(* POU Device/Valve/fbWaterSupplyValve, ST *)
FUNCTION_BLOCK fbWaterSupplyValve
VAR_INPUT
	xManualMode:			BOOL;
	wOffDelay:				WORD:=3;
	xStopSupplying:		BOOL;
	rWaterLevel:			REAL;
	rWaterLevelNotOK:	REAL;
	xUpperLevel:			BOOL;
	xOnAutoWorking:		BOOL;
	xSensor:				BOOL;
END_VAR
VAR_IN_OUT

	xOnManual:			BOOL;

END_VAR
VAR_OUTPUT
	xDO_On:				BOOL;
	xState:					BOOL;
END_VAR
VAR
	tfOffDelay:				TOF;
	xDO_OnOld:			BOOL;
	tnDelayState:			TON;
	rtLevelDown:			R_TRIG;
	xOnAuto:				BOOL;
END_VAR
IF xManualMode THEN
	tfOffDelay(IN:=xOnManual, PT:= WORD_TO_TIME(wOffDelay * 1000), Q=>xDO_On);
ELSIF xOnAutoWorking THEN
	rtLevelDown(CLK:= rWaterLevel < rWaterLevelNotOK);
	IF rWaterLevel < rWaterLevelNotOK THEN
		xOnAuto:=TRUE;
	END_IF
	IF xUpperLevel THEN
		xOnAuto:=FALSE;
	END_IF

	tfOffDelay(IN:=xOnAuto, PT:= WORD_TO_TIME(wOffDelay * 1000), Q=>xDO_On);
END_IF

xState:=xSensor;

IF xStopSupplying THEN
	xDO_On:=FALSE;
END_IF
(*
IF NOT xOnAutoWorking THEN
	xDO_On:=FALSE;
END_IF
*)
(*
IF xDO_OnOld <> xDO_On THEN
	tnDelayState(IN:=TRUE, PT:=T#3S);
	IF tnDelayState.Q THEN
		xState:= 		xDO_On;
		xDO_OnOld:=	xDO_On;
		tnDelayState(IN:=FALSE);
	END_IF
END_IF
*)
END_FUNCTION_BLOCK

(* POU Process/prProcess, ST *)
PROGRAM prProcess
VAR
END_VAR
prDissolvingProcess();
(*
prSelfWashing();
*)
prRecipe();
prWashingProcess();
END_PROGRAM

(* POU Process/Dissolving/prDissolvingProcess, ST *)
PROGRAM prDissolvingProcess
VAR
	rtStart:	R_TRIG;
	ftStart:	F_TRIG;
	ftStop:	R_TRIG;
	rtAlkaliStart:	R_TRIG;
	rtAccidStart:	R_TRIG;
	ftAlkaliStart:	F_TRIG;
	ftAccidStart:	F_TRIG;
	ftAlkaliStop:	F_TRIG;
	ftAccidStop:	F_TRIG;
	ftPauseAlkAcc:	F_TRIG;
	rtPause:	R_TRIG;
	ftPause:	F_TRIG;

END_VAR
IF xDissolDoAlkali THEN
	CASE wDissolLineAlkali OF

				1:

					ftAlkaliStart(CLK:=xDissolving_StartLine1);
					IF ftAlkaliStart.Q THEN
						xStartDissolvingAlkali:=FALSE;
						xPauseDissolvingAlkali:=FALSE;
					END_IF
					xDissolving_PausetLine1:=xPauseDissolvingAlkali;
					IF SelfWashState = 0 THEN
						prDissolvingLine1();
					END_IF

				2:

					ftAlkaliStart(CLK:=xDissolving_StartLine2);
					IF ftAlkaliStart.Q THEN
						xStartDissolvingAlkali:=FALSE;
						xPauseDissolvingAlkali:=FALSE;
					END_IF
					xDissolving_PausetLine2:=xPauseDissolvingAlkali;
					prDissolvingLine2();
				3:

					ftAlkaliStart(CLK:=xDissolving_StartLine3);
					IF ftAlkaliStart.Q THEN
						xStartDissolvingAlkali:=FALSE;
						xPauseDissolvingAlkali:=FALSE;
					END_IF
					xDissolving_PausetLine3:=xPauseDissolvingAlkali;
					prDissolvingLine3();
				4:

					ftAlkaliStart(CLK:=xDissolving_StartLine4);
					IF ftAlkaliStart.Q THEN
						xStartDissolvingAlkali:=FALSE;
						xPauseDissolvingAlkali:=FALSE;
					END_IF
					xDissolving_PausetLine4:=xPauseDissolvingAlkali;
					prDissolvingLine4();

	END_CASE
END_IF

IF (wDissolLineAccid <> wDissolLineAlkali OR(NOT xDissolDoAlkali) ) AND xDissilDoAccid THEN
	CASE wDissolLineAccid OF

				1:
					prDissolvingLine1();
					ftAccidStart(CLK:=xDissolving_StartLine1);
					xDissolving_PausetLine1:=xPauseDissolvingAccid;
					IF ftAccidStart.Q THEN
						xStartDissolvingAccid:=FALSE;
						xPauseDissolvingAccid:=FALSE;
					END_IF
				2:
					prDissolvingLine2();
					ftAccidStart(CLK:=xDissolving_StartLine2);
					xDissolving_PausetLine2:=xPauseDissolvingAccid;
					IF ftAccidStart.Q THEN
						xStartDissolvingAccid:=FALSE;
						xPauseDissolvingAccid:=FALSE;
					END_IF
				3:
					prDissolvingLine3();
					ftAccidStart(CLK:=xDissolving_StartLine3);
					xDissolving_PausetLine3:=xPauseDissolvingAccid;
					IF ftAccidStart.Q THEN
						xStartDissolvingAccid:=FALSE;
						xPauseDissolvingAccid:=FALSE;
					END_IF
				4:
					prDissolvingLine4();
					ftAccidStart(CLK:=xDissolving_StartLine4);
					xDissolving_PausetLine4:=xPauseDissolvingAccid;
					IF ftAccidStart.Q THEN
						xStartDissolvingAccid:=FALSE;
						xPauseDissolvingAccid:=FALSE;
					END_IF

	END_CASE
END_IF


rtStart(CLK:=xDissolving_Start);
IF rtStart.Q THEN
	xDissolving_StartLine1:=	wWashingStateLine1 = 0 AND ((wDissolLineAccid = 1 AND xDissilDoAccid) OR (wDissolLineAlkali =1 AND xDissolDoAlkali));
	xDissolving_StartLine2:=	wWashingStateLine2 = 0 AND ((wDissolLineAccid = 2 AND xDissilDoAccid) OR (wDissolLineAlkali =2 AND xDissolDoAlkali));
	xDissolving_StartLine3:=	wWashingStateLine3 = 0 AND ((wDissolLineAccid = 3 AND xDissilDoAccid) OR (wDissolLineAlkali =3 AND xDissolDoAlkali));
	xDissolving_StartLine4:=	wWashingStateLine4 = 0 AND ((wDissolLineAccid = 4 AND xDissilDoAccid) OR (wDissolLineAlkali =4 AND xDissolDoAlkali));
	xStartDissolvingAlkali:=	xDissolDoAlkali;
	xStartDissolvingAccid:=	xDissilDoAccid;
END_IF

ftStart(CLK:=xDissolving_Start);
IF ftStart.Q THEN
	xDissolving_StartLine1:=	FALSE;
	xDissolving_StartLine2:=	FALSE;
	xDissolving_StartLine3:=	FALSE;
	xDissolving_StartLine4:=	FALSE;
	xStartDissolvingAlkali:=	FALSE;
	xStartDissolvingAccid:=	FALSE;
END_IF
(*
ftStop(CLK:=(xDissolving_StartLine1 OR xDissolving_StartLine2 OR xDissolving_StartLine3 OR xDissolving_StartLine4));

IF ftStop.Q THEN
	xDissolving_Start:=FALSE;
END_IF
*)
rtAlkaliStart(CLK:=xStartDissolvingAlkali);
IF rtAlkaliStart.Q THEN
	CASE wDissolLineAlkali OF

				1: xDissolving_StartLine1:=	wWashingStateLine1 = 0 AND xDissolDoAlkali;
				2: xDissolving_StartLine2:=	wWashingStateLine2 = 0 AND xDissolDoAlkali;
				3: xDissolving_StartLine3:=	wWashingStateLine3 = 0 AND xDissolDoAlkali;
				4: xDissolving_StartLine4:=	wWashingStateLine4 = 0 AND xDissolDoAlkali;

	END_CASE
END_IF

ftAlkaliStop(CLK:=xStartDissolvingAlkali);
IF ftAlkaliStop.Q THEN
	CASE wDissolLineAlkali OF

				1: xDissolving_StartLine1:=	FALSE;
				2: xDissolving_StartLine2:=	FALSE;
				3: xDissolving_StartLine3:=	FALSE;
				4: xDissolving_StartLine4:=	FALSE;

	END_CASE
END_IF

rtAccidStart(CLK:=xStartDissolvingAccid);
IF rtAccidStart.Q THEN
	CASE wDissolLineAccid OF

				1: xDissolving_StartLine1:=	wWashingStateLine1 = 0 AND xDissilDoAccid;
				2: xDissolving_StartLine2:=	wWashingStateLine2 = 0 AND xDissilDoAccid;
				3: xDissolving_StartLine3:=	wWashingStateLine3 = 0 AND xDissilDoAccid;
				4: xDissolving_StartLine4:=	wWashingStateLine4 = 0 AND xDissilDoAccid;

	END_CASE
END_IF

ftAccidStop(CLK:=xStartDissolvingAccid);
IF ftAccidStop.Q THEN
	CASE wDissolLineAccid OF

				1: xDissolving_StartLine1:=	FALSE;
				2: xDissolving_StartLine2:=	FALSE;
				3: xDissolving_StartLine3:=	FALSE;
				4: xDissolving_StartLine4:=	FALSE;

	END_CASE
END_IF
IF NOT(xDissolving_StartLine1 OR xDissolving_StartLine2 OR xDissolving_StartLine3 OR xDissolving_StartLine4) THEN
	xDissolving_Start:=FALSE;
END_IF
rtPause(CLK:=xDissolving_Pause);
ftPause(CLK:=xDissolving_Pause);
ftPauseAlkAcc(CLK:= xPauseDissolvingAccid OR xPauseDissolvingAlkali);

IF rtPause.Q THEN
	xPauseDissolvingAccid:=TRUE;
	xPauseDissolvingAlkali:=TRUE;
END_IF
IF ftPause.Q THEN
	xPauseDissolvingAccid:=FALSE;
	xPauseDissolvingAlkali:=FALSE;
END_IF

IF ftPauseAlkAcc.Q THEN
	xDissolving_Pause:=FALSE;
END_IF


prDissolvStateBits();
END_PROGRAM

(* POU Process/Dissolving/prDissolvingLine1, ST *)
PROGRAM prDissolvingLine1
VAR
	Dissolving1:			fbDissolving;
	xResetErrors: BOOL;
END_VAR
Dissolving1(
					xDoAccid:=xDissilDoAccid AND wDissolLineAccid = 1,
					xDoAlkali:=xDissolDoAlkali AND wDissolLineAlkali =1,
					xAlkaliUpperLevel:= DI_AlkaliUpperLevel,
					xAccidUpperLevel:= DI_AccidUpperLevel,
					rConcGet:= Conc_Line1,
					xV_AlkaliInOn:= xState_V106,
					xV_AccidInOn:= xState_V107,
					xV_WaterOutOn:= xState_V101,
					xV_NotshortcutOn:= xState_V110,
					xV_OutOn:=xState_V111,
					wConcPumpTimeAlk:= rPA_WorkTime_Alk,
					wConcPumpTimeAcc:= rPA_WorkTime_Acc,

					wConcMessureTime:= rConcCheckTime,
					rAlkaliConcSet:= rDissolAlkaliConcSet,
					rWaterConcSet:= rDissolWaterConcSet,
					rAccidConcSet:= rDissolAccidConcSet,

					rAlkaliLevelSet:= rDissolAlkaliLevelSet,
					rAccidLevelSet:= rDissolAccidLevelSet,
					rAlkaliLevelGet:= AlkaliLevel,
					rAccidLevelGet:=AccidLevel,

					xStart:= xDissolving_StartLine1,
					(*xAccidIsGoing:= xAccidIsGoing1,*)
					xPause:=xDissolving_PausetLine1,
					xVout:= OnAuto_V111,
					xV_Notshortcut:= OnAuto_V110,
					xV_WaterOut:= OnAuto_V101,
					xV_Cycle:= OnAuto_V105,
					xV_Drainage:= OnAuto_V109,
					xV_AlkaliOut:= OnAuto_V104,
					xV_AccidOut:= OnAuto_V103,
					xV_AlkaliIn:= OnAuto_V106,
					xV_AccidIn:= OnAuto_V107,
					xPump:= Pump_OnAuto_1,
					xResetErrors:= xResetErrors,
					xPA_Alkali:= PA_OnAuto_12,
					xPA_Accid:= PA_OnAuto_11,
					wPumpFlawSet:= wFlawDissolving,
					wPumpFlawOut:= Pump_FlawAutoSet_1,
					xAlkaliIsReady:= xAlkaliIsReady,
					xAccidIsReady:= xAccidIsReady,
					State=> wDissolvingStateLine1,
					PauseState=>(*wDissolvingPauseStateLine1*),
					wError=> wDissolvingError);
END_PROGRAM

(* POU Process/Dissolving/fbDissolving, ST *)
FUNCTION_BLOCK fbDissolving
VAR_INPUT

	xDoAccid:					BOOL;
	xDoAlkali:					BOOL;
	xAlkaliUpperLevel:		BOOL;
	xAccidUpperLevel:		BOOL;
	rConcGet:					REAL;
	xV_AlkaliInOn:				BOOL;
	xV_AccidInOn:				BOOL;
	xV_WaterOutOn:			BOOL;
	xV_NotshortcutOn:		BOOL;
	xV_OutOn:					BOOL;

	rAlkaliConcSet: 			REAL;
	rWaterConcSet:			REAL;
	rAccidConcSet:			REAL;
	wConcPumpTimeAlk:		WORD:=60;
	wConcPumpTimeAcc:	WORD:=300;
	wConcMessureTime:		WORD:=5;
	wPumpFlawSet:			REAL;
	xPause:					BOOL;
	rAlkaliLevelSet:			REAL;
	rAccidLevelSet:			REAL;
	rAlkaliLevelGet:			REAL;
	rAccidLevelGet:			REAL;


END_VAR
VAR_IN_OUT

	xStart:						BOOL;
	xVout:						BOOL;
	xV_Notshortcut:			BOOL;
	xV_WaterOut:				BOOL;
	xV_Cycle:					BOOL;
	xV_Drainage:				BOOL;
	xV_AlkaliOut:				BOOL;
	xV_AccidOut:				BOOL;
	xV_AlkaliIn:				BOOL;
	xV_AccidIn:				BOOL;

	xPump:					BOOL;
	xResetErrors:				BOOL;
	xPA_Alkali:					BOOL;
	xPA_Accid:					BOOL;
	wPumpFlawOut:			REAL;

	xAlkaliIsReady:			BOOL;
	xAccidIsReady:			BOOL;


END_VAR


VAR_OUTPUT

	State:					Dissolving_States;
	PauseState:			Dissolving_States;
	wError:					WORD;


END_VAR
VAR
	rtStart:					R_TRIG;
	rtPause:				R_TRIG;
	ftStart:					F_TRIG;
	tnWaitErr:				TON;
	tnConc:				TON;
	tnPA:					TON;
	xAccidIsGoing:			BOOL;


END_VAR
rtStart(CLK:=xStart);
ftStart(CLK:=xStart);
rtPause(CLK:=xPause);


IF rtStart.Q THEN
	xAlkaliIsReady:=NOT xDoAlkali;
	xAccidIsReady:=NOT xDoAccid;
	wPumpFlawOut:=wPumpFlawSet;
	tnConc(IN:=FALSE);
	tnPA(IN:=FALSE);
	xPause:=	FALSE;
	State:=WaterStart;
END_IF

IF ftStart.Q THEN
	wError:=0;
	xVout:=					FALSE;
	xV_Notshortcut:=		FALSE;

	xV_AlkaliIn:=			FALSE;
	xV_AccidIn:=			FALSE;
	xV_WaterOut:=		FALSE;
	xV_AlkaliOut:=			FALSE;
	xV_AccidOut:=			FALSE;
	xV_Cycle:=				FALSE;
	xV_Drainage:=		FALSE;
	xPump:=				FALSE;
	xPA_Alkali:= 			FALSE;
	xPA_Accid:=			FALSE;
	xPause:=				FALSE;
	State:=					DissolvingStop;
END_IF

IF rtPause.Q THEN
	PauseState:=State;
	xPump:= FALSE;
	xPA_Alkali:= FALSE;
	xPA_Accid:=FALSE;
	State:=DissolvingPause;
END_IF

CASE State OF



			DissolvingStop:
							;


			DissolvingPause:

				IF NOT xPause THEN
					State:= PauseState;
				END_IF



			WaterStart:

				xV_Notshortcut:=		FALSE;
				xVout:= 				FALSE;

				tnWaitErr(IN:= (xV_NotshortcutOn OR xV_OutOn), PT:=T#20S);
				IF tnWaitErr.Q THEN
					wError.0:=TRUE;
				END_IF
				xPump:= TRUE;
				IF NOT (xV_NotshortcutOn OR xV_OutOn) THEN
					IF xDoAlkali THEN
						State:=AlkaliTankFullUp;
					ELSIF xDoAccid THEN
						State:=AccidTankFullUp;
					END_IF
				END_IF



			AlkaliTankFullUp:


				IF rAlkaliLevelGet > rAlkaliLevelSet THEN
					State:=AlkaliConc;
				END_IF

				IF NOT (xV_NotshortcutOn OR xV_OutOn) THEN
					xV_WaterOut:= 	TRUE;
					xV_AlkaliIn:=		TRUE;
					xV_Drainage:=	TRUE;
				END_IF


				IF xV_AlkaliInOn AND xV_WaterOutOn THEN
					xPump:=TRUE;
				END_IF




			AlkaliConc:

				xAccidIsGoing:=	FALSE;
				xV_WaterOut:= 	FALSE;
				xV_AlkaliOut:=		TRUE;
				xV_AlkaliIn:=		TRUE;
				xPA_Alkali:=		TRUE;
				xPump:=TRUE;

				tnPA(IN:=xPA_Alkali, PT:= (WORD_TO_TIME(wConcPumpTimeAlk)*1000));
				IF tnPA.Q THEN
					xPA_Alkali:=FALSE;
					tnPA(IN:=FALSE);
					State:= AlkaliConcMessure;
				END_IF



			AlkaliConcMessure:

				xPump:=TRUE;
				tnConc(IN:= TRUE, PT:=(WORD_TO_TIME(wConcMessureTime)*1000));
				IF tnConc.Q THEN
					tnConc(IN:= FALSE);
					IF rAlkaliConcSet  <  rConcGet THEN
						xAlkaliIsReady:=TRUE;
						State:= WaterAfter;
					ELSE
						xAlkaliIsReady:=FALSE;
						State:= AlkaliConc;
					END_IF
				END_IF



			WaterAfter:


				xV_AlkaliIn:=		FALSE;
				xV_AccidIn:=		FALSE;
				xV_Drainage:=	FALSE;
				xV_AlkaliOut:=		FALSE;
				xV_AccidOut:=		FALSE;
				xV_WaterOut:= 	TRUE;
				xPump:=			TRUE;

				tnConc(IN:=  rConcGet < 0.1, PT:=T#80S);
				IF tnConc.Q THEN
					tnConc(IN:=FALSE);
					IF xAccidIsReady OR (NOT xDoAccid) THEN
						xStart:=FALSE;
					ELSIF xDoAccid THEN
						State:= AccidTankFullUp;
					END_IF
				END_IF


			AccidTankFullUp:


				IF rAccidLevelGet > rAccidLevelSet THEN
					State:=AccidConc;
				END_IF

				IF NOT (xV_NotshortcutOn OR xV_OutOn) THEN
					xV_WaterOut:= 	TRUE;
					xV_AccidIn:=		TRUE;
					xV_Drainage:=	TRUE;
				END_IF

				IF xV_AccidInOn AND xV_WaterOutOn THEN
					xPump:=TRUE;
				END_IF




			AccidConc:

				xAccidIsGoing:=	TRUE;
				xV_WaterOut:= 	FALSE;
				xV_AccidOut:=		TRUE;
				xV_AccidIn:=		TRUE;
				xPA_Accid:=		TRUE;
				xV_Drainage:=	TRUE;
				xPump:=			TRUE;

				tnPA(IN:=xPA_Accid, PT:= (WORD_TO_TIME(wConcPumpTimeAcc)*1000));
				IF tnPA.Q THEN
					xPA_Accid:=FALSE;
					tnPA(IN:=FALSE);
					State:= AccidConcMessure;
				END_IF





		AccidConcMessure:

				xPump:=TRUE;
				tnConc(IN:= TRUE, PT:=(WORD_TO_TIME(wConcMessureTime)*1000));
				IF tnConc.Q THEN
					tnConc(IN:= FALSE);
					IF rAccidConcSet  <  rConcGet THEN
						xAccidIsReady:=TRUE;
						State:= WaterAfter;
					ELSE
						xAccidIsReady:=FALSE;
						State:= AccidConc;
					END_IF
				END_IF


END_CASE
END_FUNCTION_BLOCK

(* POU Process/Dissolving/prDissolvingLine2, ST *)
PROGRAM prDissolvingLine2
VAR
	Dissolving2:			fbDissolving;
	xResetErrors: BOOL;
END_VAR
IF wWashingStateLine2 = 0 THEN
Dissolving2(
					xDoAccid:=xDissilDoAccid AND wDissolLineAccid = 2,
					xDoAlkali:=xDissolDoAlkali AND wDissolLineAlkali =2,
					xAlkaliUpperLevel:= DI_AlkaliUpperLevel,
					xAccidUpperLevel:= DI_AccidUpperLevel,
					rConcGet:= Conc_Line2,
					xV_AlkaliInOn:= xState_V206,
					xV_AccidInOn:= xState_V207,
					xV_WaterOutOn:= xState_V201,
					xV_NotshortcutOn:= xState_V210,
					xV_OutOn:=xState_V211,
					wConcPumpTimeAlk:= rPA_WorkTime_Alk,
					wConcPumpTimeAcc:= rPA_WorkTime_Acc,
					wConcMessureTime:= rConcCheckTime,
					rAlkaliConcSet:= rDissolAlkaliConcSet,
					rWaterConcSet:= rDissolWaterConcSet,
					rAccidConcSet:= rDissolAccidConcSet,

					rAlkaliLevelSet:= rDissolAlkaliLevelSet,
					rAccidLevelSet:= rDissolAccidLevelSet,
					rAlkaliLevelGet:= AlkaliLevel,
					rAccidLevelGet:=AccidLevel,

					xStart:= xDissolving_StartLine2,
					(*xAccidIsGoing:= xAccidIsGoing2,*)
					xPause:=xDissolving_PausetLine2,
					xVout:= OnAuto_V211,
					xV_Notshortcut:= OnAuto_V210,
					xV_WaterOut:= OnAuto_V201,
					xV_Cycle:= OnAuto_V205,
					xV_Drainage:= OnAuto_V209,
					xV_AlkaliOut:= OnAuto_V204,
					xV_AccidOut:= OnAuto_V203,
					xV_AlkaliIn:= OnAuto_V206,
					xV_AccidIn:= OnAuto_V207,
					xPump:= Pump_OnAuto_2,
					xResetErrors:= xResetErrors,
					xPA_Alkali:= PA_OnAuto_12,
					xPA_Accid:= PA_OnAuto_11,
					wPumpFlawSet:= wFlawDissolving,
					wPumpFlawOut:= Pump_FlawAutoSet_2,
					xAlkaliIsReady:= xAlkaliIsReady,
					xAccidIsReady:= xAccidIsReady,
					State=> wDissolvingStateLine2,
					PauseState=>(*wDissolvingPauseStateLine2*),
					wError=> wDissolvingError);
END_IF
END_PROGRAM

(* POU Process/Dissolving/prDissolvingLine3, ST *)
PROGRAM prDissolvingLine3
VAR
	Dissolving3:			fbDissolving;
	xResetErrors: BOOL;
END_VAR
IF wWashingStateLine3 = 0 THEN
Dissolving3(
					xDoAccid:=xDissilDoAccid AND wDissolLineAccid = 3,
					xDoAlkali:=xDissolDoAlkali AND wDissolLineAlkali =3,
					xAlkaliUpperLevel:= DI_AlkaliUpperLevel,
					xAccidUpperLevel:= DI_AccidUpperLevel,
					rConcGet:= Conc_Line3,
					xV_AlkaliInOn:= xState_V306,
					xV_AccidInOn:= xState_V307,
					xV_WaterOutOn:= xState_V301,
					xV_NotshortcutOn:= xState_V310,
					xV_OutOn:=xState_V311,
					wConcPumpTimeAlk:= rPA_WorkTime_Alk,
					wConcPumpTimeAcc:= rPA_WorkTime_Acc,
					wConcMessureTime:= rConcCheckTime,
					rAlkaliConcSet:= rDissolAlkaliConcSet,
					rWaterConcSet:= rDissolWaterConcSet,
					rAccidConcSet:= rDissolAccidConcSet,

					rAlkaliLevelSet:= rDissolAlkaliLevelSet,
					rAccidLevelSet:= rDissolAccidLevelSet,
					rAlkaliLevelGet:= AlkaliLevel,
					rAccidLevelGet:=AccidLevel,

					xStart:= xDissolving_StartLine3,
					(*xAccidIsGoing:= xAccidIsGoing3,*)
					xPause:=xDissolving_PausetLine3,
					xVout:= OnAuto_V311,
					xV_Notshortcut:= OnAuto_V310,
					xV_WaterOut:= OnAuto_V301,
					xV_Cycle:= OnAuto_V305,
					xV_Drainage:= OnAuto_V309,
					xV_AlkaliOut:= OnAuto_V304,
					xV_AccidOut:= OnAuto_V303,
					xV_AlkaliIn:= OnAuto_V306,
					xV_AccidIn:= OnAuto_V307,
					xPump:= Pump_OnAuto_3,
					xResetErrors:= xResetErrors,
					xPA_Alkali:= PA_OnAuto_12,
					xPA_Accid:= PA_OnAuto_11,
					wPumpFlawSet:= wFlawDissolving,
					wPumpFlawOut:= Pump_FlawAutoSet_3,
					xAlkaliIsReady:= xAlkaliIsReady,
					xAccidIsReady:= xAccidIsReady,
					State=> wDissolvingStateLine3,
					PauseState=>(*wDissolvingPauseStateLine3*),
					wError=> wDissolvingError);
END_IF
END_PROGRAM

(* POU Process/Dissolving/prDissolvingLine4, ST *)
PROGRAM prDissolvingLine4
VAR
	Dissolving4:			fbDissolving;
	xResetErrors: BOOL;
END_VAR
IF wWashingStateLine4 = 0 THEN
Dissolving4(
					xDoAccid:=xDissilDoAccid AND wDissolLineAccid = 4,
					xDoAlkali:=xDissolDoAlkali AND wDissolLineAlkali =4,
					xAlkaliUpperLevel:= DI_AlkaliUpperLevel,
					xAccidUpperLevel:= DI_AccidUpperLevel,
					rConcGet:= Conc_Line4,
					xV_AlkaliInOn:= xState_V406,
					xV_AccidInOn:= xState_V407,
					xV_WaterOutOn:= xState_V401,
					xV_NotshortcutOn:= xState_V410,
					xV_OutOn:=xState_V411,
					wConcPumpTimeAlk:= rPA_WorkTime_Alk,
					wConcPumpTimeAcc:= rPA_WorkTime_Acc,
					wConcMessureTime:= rConcCheckTime,
					rAlkaliConcSet:= rDissolAlkaliConcSet,
					rWaterConcSet:= rDissolWaterConcSet,
					rAccidConcSet:= rDissolAccidConcSet,

					rAlkaliLevelSet:= rDissolAlkaliLevelSet,
					rAccidLevelSet:= rDissolAccidLevelSet,
					rAlkaliLevelGet:= AlkaliLevel,
					rAccidLevelGet:=AccidLevel,

					xStart:= xDissolving_StartLine4,
					(*xAccidIsGoing:= xAccidIsGoing4,*)
					xPause:=xDissolving_PausetLine4,
					xVout:= OnAuto_V411,
					xV_Notshortcut:= OnAuto_V410,
					xV_WaterOut:= OnAuto_V401,
					xV_Cycle:= OnAuto_V405,
					xV_Drainage:= OnAuto_V409,
					xV_AlkaliOut:= OnAuto_V404,
					xV_AccidOut:= OnAuto_V403,
					xV_AlkaliIn:= OnAuto_V406,
					xV_AccidIn:= OnAuto_V407,
					xPump:= Pump_OnAuto_4,
					xResetErrors:= xResetErrors,
					xPA_Alkali:= PA_OnAuto_12,
					xPA_Accid:= PA_OnAuto_11,
					wPumpFlawSet:= wFlawDissolving,
					wPumpFlawOut:= Pump_FlawAutoSet_4,
					xAlkaliIsReady:= xAlkaliIsReady,
					xAccidIsReady:= xAccidIsReady,
					State=> wDissolvingStateLine4,
					PauseState=>(*wDissolvingPauseStateLine4*),
					wError=> wDissolvingError);
END_IF
END_PROGRAM

(* POU Process/Dissolving/prDissolvStateBits, ST *)
PROGRAM prDissolvStateBits
VAR
END_VAR
wDissolvingStateBitsLine1.0	:=	wDissolvingStateLine1 = 0	;
wDissolvingStateBitsLine1.1	:=	wDissolvingStateLine1 = 1	;
wDissolvingStateBitsLine1.2	:=	wDissolvingStateLine1 = 2	;
wDissolvingStateBitsLine1.3	:=	wDissolvingStateLine1 = 3	;
wDissolvingStateBitsLine1.4	:=	wDissolvingStateLine1 = 4	;
wDissolvingStateBitsLine1.5	:=	wDissolvingStateLine1 = 5	;
wDissolvingStateBitsLine1.6	:=	wDissolvingStateLine1 = 6	;
wDissolvingStateBitsLine1.7	:=	wDissolvingStateLine1 = 7	;
wDissolvingStateBitsLine1.8	:=	wDissolvingStateLine1 = 8	;
wDissolvingStateBitsLine1.9	:=	wDissolvingStateLine1 = 9	;
wDissolvingStateBitsLine1.10	:=	wDissolvingStateLine1 = 10	;
wDissolvingStateBitsLine1.11	:=	wDissolvingStateLine1 = 11	;
wDissolvingStateBitsLine1.12	:=	wDissolvingStateLine1 = 12	;
wDissolvingStateBitsLine1.13	:=	wDissolvingStateLine1 = 13	;
wDissolvingStateBitsLine1.14	:=	wDissolvingStateLine1 = 14	;
wDissolvingStateBitsLine1.15	:=	wDissolvingStateLine1 = 15	;
wDissolvingStateBitsLine1.16	:=	wDissolvingStateLine1 = 16	;
wDissolvingStateBitsLine1.17	:=	wDissolvingStateLine1 = 17	;
wDissolvingStateBitsLine1.18	:=	wDissolvingStateLine1 = 18	;
wDissolvingStateBitsLine1.19	:=	wDissolvingStateLine1 = 19	;
wDissolvingStateBitsLine1.20	:=	wDissolvingStateLine1 = 20	;
wDissolvingStateBitsLine1.21	:=	wDissolvingStateLine1 = 21	;
wDissolvingStateBitsLine1.22	:=	wDissolvingStateLine1 = 22	;
wDissolvingStateBitsLine1.23	:=	wDissolvingStateLine1 = 23	;
wDissolvingStateBitsLine1.24	:=	wDissolvingStateLine1 = 24	;
wDissolvingStateBitsLine1.25	:=	wDissolvingStateLine1 = 25	;
wDissolvingStateBitsLine1.26	:=	wDissolvingStateLine1 = 26	;
			
wDissolvingStateBitsLine2.0	:=	wDissolvingStateLine2 = 0	;
wDissolvingStateBitsLine2.1	:=	wDissolvingStateLine2 = 1	;
wDissolvingStateBitsLine2.2	:=	wDissolvingStateLine2 = 2	;
wDissolvingStateBitsLine2.3	:=	wDissolvingStateLine2 = 3	;
wDissolvingStateBitsLine2.4	:=	wDissolvingStateLine2 = 4	;
wDissolvingStateBitsLine2.5	:=	wDissolvingStateLine2 = 5	;
wDissolvingStateBitsLine2.6	:=	wDissolvingStateLine2 = 6	;
wDissolvingStateBitsLine2.7	:=	wDissolvingStateLine2 = 7	;
wDissolvingStateBitsLine2.8	:=	wDissolvingStateLine2 = 8	;
wDissolvingStateBitsLine2.9	:=	wDissolvingStateLine2 = 9	;
wDissolvingStateBitsLine2.10	:=	wDissolvingStateLine2 = 10	;
wDissolvingStateBitsLine2.11	:=	wDissolvingStateLine2 = 11	;
wDissolvingStateBitsLine2.12	:=	wDissolvingStateLine2 = 12	;
wDissolvingStateBitsLine2.13	:=	wDissolvingStateLine2 = 13	;
wDissolvingStateBitsLine2.14	:=	wDissolvingStateLine2 = 14	;
wDissolvingStateBitsLine2.15	:=	wDissolvingStateLine2 = 15	;
wDissolvingStateBitsLine2.16	:=	wDissolvingStateLine2 = 16	;
wDissolvingStateBitsLine2.17	:=	wDissolvingStateLine2 = 17	;
wDissolvingStateBitsLine2.18	:=	wDissolvingStateLine2 = 18	;
wDissolvingStateBitsLine2.19	:=	wDissolvingStateLine2 = 19	;
wDissolvingStateBitsLine2.20	:=	wDissolvingStateLine2 = 20	;
wDissolvingStateBitsLine2.21	:=	wDissolvingStateLine2 = 21	;
wDissolvingStateBitsLine2.22	:=	wDissolvingStateLine2 = 22	;
wDissolvingStateBitsLine2.23	:=	wDissolvingStateLine2 = 23	;
wDissolvingStateBitsLine2.24	:=	wDissolvingStateLine2 = 24	;
wDissolvingStateBitsLine2.25	:=	wDissolvingStateLine2 = 25	;
wDissolvingStateBitsLine2.26	:=	wDissolvingStateLine2 = 26	;
			
wDissolvingStateBitsLine3.0	:=	wDissolvingStateLine3 = 0	;
wDissolvingStateBitsLine3.1	:=	wDissolvingStateLine3 = 1	;
wDissolvingStateBitsLine3.2	:=	wDissolvingStateLine3 = 2	;
wDissolvingStateBitsLine3.3	:=	wDissolvingStateLine3 = 3	;
wDissolvingStateBitsLine3.4	:=	wDissolvingStateLine3 = 4	;
wDissolvingStateBitsLine3.5	:=	wDissolvingStateLine3 = 5	;
wDissolvingStateBitsLine3.6	:=	wDissolvingStateLine3 = 6	;
wDissolvingStateBitsLine3.7	:=	wDissolvingStateLine3 = 7	;
wDissolvingStateBitsLine3.8	:=	wDissolvingStateLine3 = 8	;
wDissolvingStateBitsLine3.9	:=	wDissolvingStateLine3 = 9	;
wDissolvingStateBitsLine3.10	:=	wDissolvingStateLine3 = 10	;
wDissolvingStateBitsLine3.11	:=	wDissolvingStateLine3 = 11	;
wDissolvingStateBitsLine3.12	:=	wDissolvingStateLine3 = 12	;
wDissolvingStateBitsLine3.13	:=	wDissolvingStateLine3 = 13	;
wDissolvingStateBitsLine3.14	:=	wDissolvingStateLine3 = 14	;
wDissolvingStateBitsLine3.15	:=	wDissolvingStateLine3 = 15	;
wDissolvingStateBitsLine3.16	:=	wDissolvingStateLine3 = 16	;
wDissolvingStateBitsLine3.17	:=	wDissolvingStateLine3 = 17	;
wDissolvingStateBitsLine3.18	:=	wDissolvingStateLine3 = 18	;
wDissolvingStateBitsLine3.19	:=	wDissolvingStateLine3 = 19	;
wDissolvingStateBitsLine3.20	:=	wDissolvingStateLine3 = 20	;
wDissolvingStateBitsLine3.21	:=	wDissolvingStateLine3 = 21	;
wDissolvingStateBitsLine3.22	:=	wDissolvingStateLine3 = 22	;
wDissolvingStateBitsLine3.23	:=	wDissolvingStateLine3 = 23	;
wDissolvingStateBitsLine3.24	:=	wDissolvingStateLine3 = 24	;
wDissolvingStateBitsLine3.25	:=	wDissolvingStateLine3 = 25	;
wDissolvingStateBitsLine3.26	:=	wDissolvingStateLine3 = 26	;
			
wDissolvingStateBitsLine4.0	:=	wDissolvingStateLine4 = 0	;
wDissolvingStateBitsLine4.1	:=	wDissolvingStateLine4 = 1	;
wDissolvingStateBitsLine4.2	:=	wDissolvingStateLine4 = 2	;
wDissolvingStateBitsLine4.3	:=	wDissolvingStateLine4 = 3	;
wDissolvingStateBitsLine4.4	:=	wDissolvingStateLine4 = 4	;
wDissolvingStateBitsLine4.5	:=	wDissolvingStateLine4 = 5	;
wDissolvingStateBitsLine4.6	:=	wDissolvingStateLine4 = 6	;
wDissolvingStateBitsLine4.7	:=	wDissolvingStateLine4 = 7	;
wDissolvingStateBitsLine4.8	:=	wDissolvingStateLine4 = 8	;
wDissolvingStateBitsLine4.9	:=	wDissolvingStateLine4 = 9	;
wDissolvingStateBitsLine4.10	:=	wDissolvingStateLine4 = 10	;
wDissolvingStateBitsLine4.11	:=	wDissolvingStateLine4 = 11	;
wDissolvingStateBitsLine4.12	:=	wDissolvingStateLine4 = 12	;
wDissolvingStateBitsLine4.13	:=	wDissolvingStateLine4 = 13	;
wDissolvingStateBitsLine4.14	:=	wDissolvingStateLine4 = 14	;
wDissolvingStateBitsLine4.15	:=	wDissolvingStateLine4 = 15	;
wDissolvingStateBitsLine4.16	:=	wDissolvingStateLine4 = 16	;
wDissolvingStateBitsLine4.17	:=	wDissolvingStateLine4 = 17	;
wDissolvingStateBitsLine4.18	:=	wDissolvingStateLine4 = 18	;
wDissolvingStateBitsLine4.19	:=	wDissolvingStateLine4 = 19	;
wDissolvingStateBitsLine4.20	:=	wDissolvingStateLine4 = 20	;
wDissolvingStateBitsLine4.21	:=	wDissolvingStateLine4 = 21	;
wDissolvingStateBitsLine4.22	:=	wDissolvingStateLine4 = 22	;
wDissolvingStateBitsLine4.23	:=	wDissolvingStateLine4 = 23	;
wDissolvingStateBitsLine4.24	:=	wDissolvingStateLine4 = 24	;
wDissolvingStateBitsLine4.25	:=	wDissolvingStateLine4 = 25	;
wDissolvingStateBitsLine4.26	:=	wDissolvingStateLine4 = 26	;
END_PROGRAM

(* POU Process/Recipe/prRecipe, ST *)
PROGRAM prRecipe
VAR
	RecipeOperate:	fbRecipeOperate;
END_VAR
wLine:=1;
RecipeOperate(
	wLine:= wLine,
	wRecipe:= wRecipe,
	xSave:= xSave,
	arAlkaliTime:= 	arAlkaliTime,
	arTalkaliSet:= 	arTalkaliSet,
	arFlawAlkaliSet:= 	arFlawAlkaliSet, 
	arConcAlkaliSet:= 	arConcAlkaliSet,
	arAccidTime:= 	arAccidTime, 
	arTaccidSet:= 	arTaccidSet,
	arFlawAccidSet:= 	arFlawAccidSet, 
	arConcAccidSet:= 	arConcAccidSet, 
	arWaterTime:= 	arWaterTime,
	arTwaterSet:= 	arTwaterSet, 
	arFlawWaterSet:=	arFlawWaterSet,
	arAfterAccidWaterTime:= 	arAfterAccidWaterTime, 
	arTafterAccidWater:= 	arTafterAccidWater, 
	arConcAfterAccidWaterSet:= 	arConcAfterAccidWaterSet,
	arAfterAlkaliWaterTime:= 	arAfterAlkaliWaterTime,
	arTafterAlkaliWater:= 	arTafterAlkaliWater,
	arConcAfterAlkaliWaterSet:= 	arConcAfterAlkaliWaterSet,
	arTsterilSet:= 	arTsterilSet, 
	arFlawSterilSet:= 	arFlawSterilSet,
	arConcSterilSet:= 	arConcSterilSet,
	arSterilTime:= 	arSterilTime,
	arFlawWaterAfterAlcaliSet:=	arFlawWaterAfterAlcaliSet,
	arFlawWaterAfterAccidSet:=	arFlawWaterAfterAccidSet,
	arWaterAfterSterilFlaw:=	arWaterAfterSterilFlaw,
	arWaterAfterSterilConc:=	arWaterAfterSterilConc,
	arWaterAfterSterilT:=	arWaterAfterSterilT,
	arWaterAfterSterilTime:=	arWaterAfterSterilTime,
	arConcPumpTimeSteril:= arConcPumpTimeSteril,
	wAlkaliTime:= 	wAlkaliTime,
	wTalkaliSet:= 	wTalkaliSet,
	wFlawAlkaliSet:= 	wFlawAlkaliSet,
	wConcAlkaliSet:= 	wConcAlkaliSet,
	wAccidTime:= 	wAccidTime, 
	wTaccidSet:= 	wTaccidSet,
	wFlawAccidSet:= 	wFlawAccidSet, 
	wConcAccidSet:= 	wConcAccidSet, 
	wWaterTime:= 	wWaterTime, 
	wTwaterSet:= 	wTwaterSet, 
	wFlawWaterSet:= 	wFlawWaterSet,
	wAfterAccidWaterTime:= 	wAfterAccidWaterTime, 
	wTafterAccidWater:= 	wTafterAccidWater, 
	wConcAfterAccidWaterSet:= 	wConcAfterAccidWaterSet, 
	wAfterAlkaliWaterTime:= 	wAfterAlkaliWaterTime, 
	wTafterAlkaliWater:= 	wTafterAlkaliWater, 
	wConcAfterAlkaliWaterSet:= 	wConcAfterAlkaliWaterSet, 
	wTsteril:= 	wTsteril,
	rFlawWaterAfterAlcaliSet:=	rFlawWaterAfterAlcaliSet,
	rFlawWaterAfterAccidSet:=	rFlawWaterAfterAccidSet,
	wConcPumpTimeSteril:=wConcPumpTimeSteril,
	wFlawSteril:= 	wFlawSteril,
	rConcSteril:= 	rConcSteril,
	wSterilTime:= 	wSterilTime,

	rWaterAfterSterilFlaw:= 	rWaterAfterSterilFlaw,
	rWaterAfterSterilConc:= 	rWaterAfterSterilConc,
	rWaterAfterSterilT:= 	rWaterAfterSterilT,
	rWaterAfterSterilTime:= 	rWaterAfterSterilTime,
	arOperations=> arOperations,
	arOperations2x=>arOperations2x,
	arOperations3x=>arOperations3x);
END_PROGRAM

(* POU Process/Recipe/fbRecipeOperate, ST *)
FUNCTION_BLOCK fbRecipeOperate
VAR_INPUT

	wLine:							WORD;
	wRecipe:						WORD;


END_VAR

VAR_IN_OUT
	xSave:							BOOL;
	arAlkaliTime:					ARRAY[1..4, 1..10] OF WORD;
	arTalkaliSet: 					ARRAY[1..4, 1..10] OF WORD;
	arFlawAlkaliSet: 				ARRAY[1..4, 1..10] OF REAL;
	arConcAlkaliSet: 				ARRAY[1..4, 1..10] OF REAL;

	arAccidTime:					ARRAY[1..4, 1..10] OF WORD;
	arTaccidSet: 					ARRAY[1..4, 1..10] OF WORD;
	arFlawAccidSet: 				ARRAY[1..4, 1..10] OF REAL;
	arConcAccidSet:				ARRAY[1..4, 1..10] OF REAL;

	arWaterTime: 					ARRAY[1..4, 1..10] OF WORD;
	arTwaterSet: 					ARRAY[1..4, 1..10] OF WORD;
	arFlawWaterSet: 				ARRAY[1..4, 1..10] OF REAL;

	arAfterAccidWaterTime: 		ARRAY[1..4, 1..10] OF WORD;
	arTafterAccidWater: 			ARRAY[1..4, 1..10] OF WORD;
	arConcAfterAccidWaterSet: 	ARRAY[1..4, 1..10] OF REAL;

	arAfterAlkaliWaterTime: 		ARRAY[1..4, 1..10] OF WORD;
	arTafterAlkaliWater: 			ARRAY[1..4, 1..10] OF WORD;
	arConcAfterAlkaliWaterSet: 	ARRAY[1..4, 1..10] OF REAL;

	arTsterilSet: 					ARRAY[1..4, 1..10] OF WORD;
	arFlawSterilSet: 				ARRAY[1..4, 1..10] OF REAL;
	arConcSterilSet: 				ARRAY[1..4, 1..10] OF REAL;
	arSterilTime: 					ARRAY[1..4, 1..10] OF WORD;

	arFlawWaterAfterAlcaliSet:	ARRAY[1..4, 1..10] OF REAL;
	arFlawWaterAfterAccidSet:	ARRAY[1..4, 1..10] OF REAL;

	arWaterAfterSterilFlaw:		ARRAY[1..4, 1..10] OF REAL;
	arWaterAfterSterilConc:		ARRAY[1..4, 1..10] OF REAL;
	arWaterAfterSterilT:			ARRAY[1..4, 1..10] OF WORD;
	arWaterAfterSterilTime:		ARRAY[1..4, 1..10] OF WORD;
	arConcPumpTimeSteril:		ARRAY[1..4, 1..10] OF WORD;


	wAlkaliTime:					WORD;
	wTalkaliSet: 					WORD;
	wFlawAlkaliSet: 				REAL;
	wConcAlkaliSet: 				REAL;

	wAccidTime:					WORD;
	wTaccidSet: 					WORD;
	wFlawAccidSet: 				REAL;
	wConcAccidSet:				REAL;

	wWaterTime: 					WORD;
	wTwaterSet: 					WORD;
	wFlawWaterSet: 				REAL;
		
	wAfterAccidWaterTime: 		WORD;
	wTafterAccidWater: 			WORD;
	wConcAfterAccidWaterSet: 	REAL;
		
	wAfterAlkaliWaterTime: 		WORD;
	wTafterAlkaliWater: 			WORD;
	wConcAfterAlkaliWaterSet: 	REAL;

	wTsteril:						WORD;
	wFlawSteril:					REAL;
	rConcSteril:					REAL;
	wSterilTime:					WORD;

	rFlawWaterAfterAlcaliSet:		REAL;
	rFlawWaterAfterAccidSet:		REAL;

	rWaterAfterSterilFlaw:			REAL;
	rWaterAfterSterilConc:		REAL;
	rWaterAfterSterilT:				WORD;
	rWaterAfterSterilTime:			WORD;
	wConcPumpTimeSteril:		WORD;

END_VAR

VAR_OUTPUT
	arOperations:					ARRAY[0..7] OF BOOL;
	arOperations2x:					ARRAY[1..4,0..7] OF BOOL;
	arOperations3x:				ARRAY[1..4,1..10,0..7] OF BOOL;
END_VAR
VAR
	wLineOld:						WORD;
	wRecipeOld:					WORD;
END_VAR
IF (wLine <> wLineOld) OR (wRecipe <> wRecipeOld) THEN
	wLineOld:=wLine;
	wRecipeOld:=wRecipe;

	wAlkaliTime:=				arAlkaliTime[wLine, wRecipe];
	wTalkaliSet:= 				arTalkaliSet[wLine, wRecipe];
	wFlawAlkaliSet:= 			arFlawAlkaliSet[wLine, wRecipe];
	wConcAlkaliSet:= 			arConcAlkaliSet[wLine, wRecipe];
		
	wAccidTime:=				arAccidTime[wLine, wRecipe];
	wTaccidSet:= 				arTaccidSet[wLine, wRecipe];
	wFlawAccidSet:= 			arFlawAccidSet[wLine, wRecipe];
	wConcAccidSet:=			arConcAccidSet[wLine, wRecipe];

	wWaterTime:= 			arWaterTime[wLine, wRecipe];
	wTwaterSet:= 				arTwaterSet[wLine, wRecipe];
	wFlawWaterSet:= 			arFlawWaterSet[wLine, wRecipe];
		
	wAfterAccidWaterTime:= 		arAfterAccidWaterTime[wLine, wRecipe];
	wTafterAccidWater:= 			arTafterAccidWater[wLine, wRecipe];
	wConcAfterAccidWaterSet:= 	arConcAfterAccidWaterSet[wLine, wRecipe];
		
	wAfterAlkaliWaterTime:= 		arAfterAlkaliWaterTime[wLine, wRecipe];
	wTafterAlkaliWater:= 			arTafterAlkaliWater[wLine, wRecipe];
	wConcAfterAlkaliWaterSet:= 	arConcAfterAlkaliWaterSet[wLine, wRecipe];

	wTsteril:=						arTsterilSet[wLine, wRecipe];
	wFlawSteril:=					arFlawSterilSet[wLine, wRecipe];
	rConcSteril:=					arConcSterilSet[wLine, wRecipe];
	wSterilTime:=					arSterilTime[wLine, wRecipe];

	rFlawWaterAfterAlcaliSet:=					arFlawWaterAfterAlcaliSet[wLine, wRecipe];
	rFlawWaterAfterAccidSet:=					arFlawWaterAfterAccidSet[wLine, wRecipe];

	rWaterAfterSterilFlaw:=					arWaterAfterSterilFlaw[wLine, wRecipe];
	rWaterAfterSterilConc:=					arWaterAfterSterilConc[wLine, wRecipe];
	rWaterAfterSterilT:=						arWaterAfterSterilT[wLine, wRecipe];
	rWaterAfterSterilTime:=					arWaterAfterSterilTime[wLine, wRecipe];
	wConcPumpTimeSteril:=					arConcPumpTimeSteril[wLine, wRecipe];



END_IF

IF xSave THEN
	xSave:=FALSE;

	arAlkaliTime[wLine, wRecipe]:=				wAlkaliTime;
	arTalkaliSet[wLine, wRecipe]:= 				wTalkaliSet;
	arFlawAlkaliSet[wLine, wRecipe]:= 			wFlawAlkaliSet;
	arConcAlkaliSet[wLine, wRecipe]:= 			wConcAlkaliSet;

	arAccidTime[wLine, wRecipe]:=				wAccidTime;
	arTaccidSet[wLine, wRecipe]:= 				wTaccidSet;
	arFlawAccidSet[wLine, wRecipe]:= 			wFlawAccidSet;
	arConcAccidSet[wLine, wRecipe]:=			wConcAccidSet;
		
	arWaterTime[wLine, wRecipe]:= 				wWaterTime;
	arTwaterSet[wLine, wRecipe]:= 				wTwaterSet;
	arFlawWaterSet[wLine, wRecipe]:= 			wFlawWaterSet;
		
	arAfterAccidWaterTime[wLine, wRecipe]:= 		wAfterAccidWaterTime;
	arTafterAccidWater[wLine, wRecipe]:= 			wTafterAccidWater;
	arConcAfterAccidWaterSet[wLine, wRecipe]:= 	wConcAfterAccidWaterSet; 
		
	arAfterAlkaliWaterTime[wLine, wRecipe]:= 		wAfterAlkaliWaterTime;
	arTafterAlkaliWater[wLine, wRecipe]:= 			wTafterAlkaliWater;
	arConcAfterAlkaliWaterSet[wLine, wRecipe]:= 	wConcAfterAlkaliWaterSet;

	arTsterilSet[wLine, wRecipe]:= 					wTsteril;
	arFlawSterilSet[wLine, wRecipe]:= 				wFlawSteril;
	arConcSterilSet[wLine, wRecipe]:= 				rConcSteril;
	arSterilTime[wLine, wRecipe]:= 					wSterilTime;

	arFlawWaterAfterAlcaliSet[wLine, wRecipe]:= 				rFlawWaterAfterAlcaliSet;
	arFlawWaterAfterAccidSet[wLine, wRecipe]:= 				rFlawWaterAfterAccidSet;

	arWaterAfterSterilFlaw[wLine, wRecipe]:= 				rWaterAfterSterilFlaw;
	arWaterAfterSterilConc[wLine, wRecipe]:= 				rWaterAfterSterilConc;
	arWaterAfterSterilT[wLine, wRecipe]:= 					rWaterAfterSterilT;
	arWaterAfterSterilTime[wLine, wRecipe]:= 				rWaterAfterSterilTime;
	arConcPumpTimeSteril[wLine, wRecipe]:= 				wConcPumpTimeSteril;

	arOperations2x[wLine,0]:= wWaterTime>0;
	arOperations2x[wLine,1]:= wAlkaliTime>0;
	arOperations2x[wLine,2]:= wAfterAlkaliWaterTime>0;
	arOperations2x[wLine,3]:= wAccidTime>0;
	arOperations2x[wLine,4]:= wAfterAccidWaterTime>0;
	arOperations2x[wLine,5]:= wSterilTime>0;
	arOperations2x[wLine,6]:= rWaterAfterSterilTime>0;
	arOperations2x[wLine,7]:= TRUE;

	arOperations3x[wLine,wRecipe,0]:= wWaterTime>0;
	arOperations3x[wLine,wRecipe,1]:= wAlkaliTime>0;
	arOperations3x[wLine,wRecipe,2]:= wAfterAlkaliWaterTime>0;
	arOperations3x[wLine,wRecipe,3]:= wAccidTime>0;
	arOperations3x[wLine,wRecipe,4]:= wAfterAccidWaterTime>0;
	arOperations3x[wLine,wRecipe,5]:= wSterilTime>0;
	arOperations3x[wLine,wRecipe,6]:= rWaterAfterSterilTime>0;
	arOperations3x[wLine,wRecipe,7]:= TRUE;


END_IF
arOperations[0]:= wWaterTime>0;
arOperations[1]:= wAlkaliTime>0;
arOperations[2]:= wAfterAlkaliWaterTime>0;
arOperations[3]:= wAccidTime>0;
arOperations[4]:= wAfterAccidWaterTime>0;
arOperations[5]:= wSterilTime>0;
arOperations[6]:= rWaterAfterSterilTime>0;
arOperations[7]:= TRUE;
END_FUNCTION_BLOCK

(* POU Process/Washing/prWashingProcess, ST *)
PROGRAM prWashingProcess
VAR


END_VAR
prWashingLine1();
(*
prWashingLine2();
prWashingLine3();
prWashingLine4();
prRemoteEquipment();
prStateBits();
*)
END_PROGRAM

(* POU Process/Washing/prWashingLine1, ST *)
PROGRAM prWashingLine1
VAR
	WashingProcess1:	fbWashingProcess;
	xResetErrors: BOOL;
END_VAR
IF SelfWashState = 0 AND wDissolvingStateLine1 = 0 THEN
WashingProcess1(
	xReady:= (*xReadyForWashing AND*) wDissolvingStateLine1 = 0,
	arOperations:= arOperations,
	rWaterLevel:= CleanWaterLevel,
	rUsedWaterLevel:= UsedWaterLevel,
	rAccidLevel:= AccidLevel,
	rAlkaliLevel:= AlkaliLevel,
	wConcPumpTime:=arConcPumpTimeSteril[1, wChosenRecipeLine1],
	wConcMessureTime:= rConcCheckTime,
	arOperations2x:=arOperations2x,
	arOperations3x:=arOperations3x,
	wChosenRecipeLine:=wChosenRecipeLine1,
	wLine:=1,
	xPumpNorm:=Pump_InvNorm_1,

	rConcOfClkaliInTank:=rDissolAlkaliConcSet,
	rConcOfAccidInTank:=rDissolAccidConcSet,

	wTafterAlkaliWater:=arTafterAlkaliWater[1, wChosenRecipeLine1],
	wTafterAccidWater:=arTafterAccidWater[1, wChosenRecipeLine1],

	rFlawWaterAfterAlcaliSet:=	arFlawWaterAfterAlcaliSet[1, wChosenRecipeLine1],
	rFlawWaterAfterAccidSet:=	arFlawWaterAfterAccidSet[1, wChosenRecipeLine1],
	rWaterAfterSterilFlaw:=	arWaterAfterSterilFlaw[1, wChosenRecipeLine1],
	rWaterAfterSterilConc:=	arWaterAfterSterilConc[1, wChosenRecipeLine1],

	rFlawWaterAfterAlcaliSet:=	arFlawWaterAfterAlcaliSet[1, wChosenRecipeLine1],
	rFlawWaterAfterAccidSet:=	arFlawWaterAfterAccidSet[1, wChosenRecipeLine1],
	wUsedWaterLevelOK:= wUsedWaterLevelOK,
	wUsedWaterLevelNotOK:= wUsedWaterLevelNotOK,
	wBackTget:=Heater_BackTget_1,
	xPause:= xPauseWashingLine1,
	xVoutOn:= xState_V104,
	xV_NotshortcutOn:= xState_V105,
	xV_AlkaliInOn:= xState_V107,
	xV_AccidInOn:= xState_V108,
	xV_WaterOutOn:= xState_V103,
	xV_AlkaliOutOn:= xState_V101,
	xV_AccidOutOn:= xState_V102,
	xV_CycleOn:= xState_V106,
	xPumpOn:= Pump_OnAuto_1,
	rConcentration:= Conc_Line1,
	(*xAccidIsGoing:=xAccidIsGoing1,*)
	xFeedbackSwitch:= DI_FeedBackSwitchLine1,
	rWaterAfterSterilT:=arWaterAfterSterilT[1, wChosenRecipeLine1],
	rWaterAfterSterilTime:=arWaterAfterSterilTime[1, wChosenRecipeLine1],
	wRecipeTimeRinse:= arWaterTime[1, wChosenRecipeLine1],
	wRecipeTimeAlcali:= arAlkaliTime[1, wChosenRecipeLine1],
	wRecipeTimeAccid:= arAccidTime[1, wChosenRecipeLine1],
	wAfterRinseConcAlk:= (*wAfterRinseConcAlk*)rConcSolutionStopoperationAlk,
	wAfterRinseConcAcc:= (*wAfterRinseConcAcc*)rConcSolutionStopoperationAcc,
	wAfterAlkWaterTime:= arAfterAlkaliWaterTime[1, wChosenRecipeLine1],
	wAfterAccWaterTime:= arAfterAccidWaterTime[1, wChosenRecipeLine1],
	rTwaterSet:= arTwaterSet[1, wChosenRecipeLine1],
	rTalcaliSet:= arTalkaliSet[1, wChosenRecipeLine1],
	rTaccidSet:= arTaccidSet[1, wChosenRecipeLine1],
	rConcAlcaliSet:= (*arConcAlkaliSet[1, wChosenRecipeLine1]*)rConcSolutionStartOperationAlk,
	rConcAccidSet:= (*arConcAccidSet[1, wChosenRecipeLine1]*)rConcSolutionStartOperationAcc,
	rFlawAlcaliSet:= arFlawAlkaliSet[1, wChosenRecipeLine1],
	rFlawWaterSet:= arFlawWaterSet[1, wChosenRecipeLine1],
	rFlawAccidSet:= arFlawAccidSet[1, wChosenRecipeLine1],
	wTsteril:= arTsterilSet[1, wChosenRecipeLine1],
	wFlawSteril:= arFlawSterilSet[1, wChosenRecipeLine1],
	rConcSteril:= arConcSterilSet[1, wChosenRecipeLine1],
	wSterilTime:= arSterilTime[1, wChosenRecipeLine1],
	wCountOfOperations:= 7,
	xStart:= xStartWashingLine1,
	xVout:= OnAuto_V104,
	xV_Notshortcut:= OnAuto_V105,
	xV_UsedWaterIn:= OnAuto_V208,
	xV_AlkaliIn:= OnAuto_V107,
	xV_AccidIn:= OnAuto_V108,
	xV_WaterOut:= OnAuto_V103,
	xV_UsedWaterOut:= OnAuto_V202,
	xV_AlkaliOut:= OnAuto_V101,
	xV_AccidOut:= OnAuto_V102,
	xV_Cycle:= OnAuto_V106,
	xV_Drainage:= OnAuto_V109,
	xPump:= Pump_OnAuto_1,
	xHeaterPower:= Heater_AutoSetT_1,
	xResetErrors:= xResetAlmAll,
	xPA:= PA_OnAuto_1,
	rToutSet:= Heater_AutoSetT_1,
	rFlawOutSet:= Pump_FlawAutoSet_1,
	xDone:=xWashingDone_Line1,
	State=> wWashingStateLine1,
	PauseState=> (*wWashingPauseStateLine1*),
	wTimePassed=> wWashingTimePassed1,
	wTimeOperationSet=> wWashingOperTimeSet1,
	wError=> wWashingErr_1);
END_IF
END_PROGRAM

(* POU Process/Washing/fbWashingProcess, ST *)
FUNCTION_BLOCK fbWashingProcess
VAR_INPUT

	xReady:						BOOL;
	arOperations:					ARRAY[0..7] OF BOOL;
	arOperations2x:				ARRAY[1..4,0..7] OF BOOL;
	arOperations3x:				ARRAY[1..4,1..10,0..7] OF BOOL;
	wLine:							WORD;
	wChosenRecipeLine:			WORD;
	rWaterLevel:					REAL;
	rUsedWaterLevel:				REAL;
	rAccidLevel:					REAL;
	rAlkaliLevel:					REAL;
	wUsedWaterLevelOK: 		REAL;
	wUsedWaterLevelNotOK: 	REAL;
	wTafterAccidWater:			WORD;
	wTafterAlkaliWater:			WORD;
	rConcOfAccidInTank:			REAL;
	rConcOfClkaliInTank:			REAL;
	xPumpNorm:					BOOL;

	wBackTget:					REAL;

	xVoutOn:						BOOL;
	xV_NotshortcutOn:			BOOL;
	xV_UsedWaterInOn:			BOOL;
	xV_AlkaliInOn:					BOOL;
	xV_AccidInOn:					BOOL;
	xV_WaterOutOn:				BOOL;
	xV_UsedWaterOutOn:			BOOL;
	xV_AlkaliOutOn:				BOOL;
	xV_AccidOutOn:				BOOL;
	xV_CycleOn:					BOOL;
	xPumpOn:						BOOL;
	rConcentration:				REAL;
	xFeedbackSwitch:				BOOL;
	wRecipeTimeRinse:			WORD;
	wRecipeTimeAlcali:			WORD;
	wRecipeTimeAccid:			WORD;
	wAfterRinseConcAlk:			REAL;
	wAfterRinseConcAcc:			REAL;
	wAfterAlkWaterTime:			WORD;
	wAfterAccWaterTime:			WORD;

	rTwaterSet:					REAL;
	rTalcaliSet:					REAL;
	rTaccidSet:					REAL;

	rConcAlcaliSet:				REAL;
	rConcAccidSet:				REAL;

	rFlawAlcaliSet:				REAL;
	rFlawWaterSet:				REAL;
	rFlawAccidSet:				REAL;

	rFlawWaterAfterAlcaliSet:		REAL;
	rFlawWaterAfterAccidSet:		REAL;

	wTsteril:						WORD;
	wFlawSteril:					REAL;
	rConcSteril:					REAL;
	wSterilTime:					WORD;
	wCountOfOperations:			WORD;
	wConcPumpTime:			WORD:=3;
	wConcMessureTime:			WORD:=5;
	rWaterAfterSterilFlaw:			REAL;
	rWaterAfterSterilConc:		REAL;
	rWaterAfterSterilT:				WORD;
	rWaterAfterSterilTime:			WORD;

END_VAR

VAR_IN_OUT
	xStart:				BOOL;
	xVout:				BOOL;
	xV_Notshortcut:		BOOL;

	xV_UsedWaterIn:	BOOL;
	xV_AlkaliIn:			BOOL;
	xV_AccidIn:			BOOL;
	
	xV_WaterOut:		BOOL;
	xV_UsedWaterOut:	BOOL;
	xV_AlkaliOut:		BOOL;
	xV_AccidOut:		BOOL;

	xV_Cycle:			BOOL;
	xV_Drainage:		BOOL;

	xPump:				BOOL;
	
	xHeaterPower:		REAL;

	xResetErrors:		BOOL;

	xPA:				BOOL;

	rToutSet:			REAL;
	rFlawOutSet:		REAL;

	xPause:						BOOL;
	xDone:				BOOL;
END_VAR

VAR_OUTPUT
	State:				WashingProcess_States;
	PauseState:		WashingProcess_States;
	wTimePassed:	WORD;
	wTimeOperationSet:	WORD;
	wError:				WORD;

END_VAR

VAR
	rtStart:				R_TRIG;
	ftStart:				F_TRIG;
	i:					WORD;
	k:					WORD;
	xRecipeNotEmpty:	BOOL;
	tnCheckWay:		TON;
	tnCheckNoFlow:		TON;
	rtCheckLevel:		R_TRIG;
	tnTimeOperation:	TON;
	xStartTimeOper:		BOOL;
	wCurrentOperation:	WORD;
	hsCheckUsedWaterLvl: HYSTERESIS;
	tnCheckConc:		TON;
	rtPause:	R_TRIG;
	PauseOperationTime:	TIME;
	tnSolutionPortion:	TON;
	xCheckConc:	BOOL;
	tnWaitConc:					TON;
	tnNoFlawErr:					TON;
	rtErrNoFlaw:					R_TRIG;
	wTimeBeforePause:			WORD;
	xCheck:	BOOL;
	xAccidIsGoing:	BOOL;
	rtPumpAlm:	R_TRIG;
	tnWaitZeroConc:	TON;

END_VAR
rtStart(CLK:=xStart);
ftStart(CLK:=xStart);
rtPause(CLK:=xPause);

IF rtStart.Q THEN
	IF xReady THEN
		xRecipeNotEmpty:=FALSE;
		wCurrentOperation:=0;
		xRecipeNotEmpty:=	FALSE;
		tnTimeOperation(IN:=FALSE);
		xDone:=FALSE;
		(*State:=FindNextOperation;*)
		State:=CheckWaterLevel;
	END_IF
END_IF


IF ftStart.Q THEN
	wError:=0;
	tnTimeOperation(IN:=FALSE);
	xVout:=					FALSE;
	xV_Notshortcut:=		FALSE;
	xV_UsedWaterIn:=	FALSE;
	xV_AlkaliIn:=			FALSE;
	xV_AccidIn:=			FALSE;
	xV_WaterOut:=		FALSE;
	xV_UsedWaterOut:=	FALSE;
	xV_AlkaliOut:=			FALSE;
	xV_AccidOut:=			FALSE;
	xV_Cycle:=				FALSE;
	xV_Drainage:=		FALSE;
	xPump:=				FALSE;
	xHeaterPower:=		0;
	xStartTimeOper:= 		FALSE;
	wCurrentOperation:=	0;
	rToutSet:=				0;
	xRecipeNotEmpty:=	FALSE;
	PauseOperationTime:=T#0S;
	wTimePassed:=		0;
	wTimeBeforePause:=0;
	wTimeOperationSet:= 0;
	xPause:=				FALSE;
	xPA:=					FALSE;
	State:=					Washing_Stop;
END_IF


IF rtPause.Q AND State > 0 THEN
	xPump:= 				FALSE;
	xPA:=					FALSE;
	rToutSet:=				0;
	wTimeBeforePause:=wTimePassed;
	PauseOperationTime:=(*PauseOperationTime + tnTimeOperation.ET*) WORD_TO_TIME(wTimePassed)*1000;
	tnTimeOperation(IN:=FALSE);

	PauseState:=State;
	State:=WashingPause;
END_IF

CASE State OF

			Washing_Stop:
								xPause:=FALSE;

			WashingPause:

				IF NOT xPause THEN
					State:= PauseState;
				END_IF




			CheckWaterLevel:


				IF rWaterLevel > rWaterLevelNotOK THEN
					State:=FindNextOperation;
				END_IF


			FindNextOperation:

				wTimePassed:=		0;
				wTimeBeforePause:=0;

				FOR i:=wCurrentOperation TO (*wCountOfOperations*)10 DO
					(*State:=i+1;*)

					IF arOperations3x[wLine,wChosenRecipeLine,i] THEN
						xRecipeNotEmpty:=	TRUE;
						wCurrentOperation:=	i+1;
						CASE i OF
							0:State:=Rinse;
							1:State:=AlkaliIn;
							2:	xV_AlkaliIn:=TRUE;
								State:=	WaterAfterAlkalin;
							3:State:=Accid;
							4:	xV_AccidIn:=TRUE;
								State:=	WaterAfterAccid;
							5:State:=Sterelisation;
							6:State:=WaterAfterSterilisation;
							7:xStart:=FALSE;
							   xDone:=TRUE;
						END_CASE
						EXIT;
					END_IF

					IF i > 7 THEN
						xStart:=FALSE;
						xDone:=TRUE;
						EXIT;
					END_IF
				END_FOR

				IF NOT (xRecipeNotEmpty AND xReady)THEN
					State:=0;
					wError.0:= NOT xReady;
					wError.1:= NOT xRecipeNotEmpty;
				END_IF


			Rinse:

				xV_Notshortcut:=	TRUE;
				xVout:= 			TRUE;
				xV_AlkaliOut:= 	FALSE;
				xV_AccidOut:= 	FALSE;
				xV_WaterOut:= 	TRUE;

				(*
				hsCheckUsedWaterLvl(
									IN:=REAL_TO_INT (rUsedWaterLevel),
									HIGH:= REAL_TO_INT(wUsedWaterLevelOK+2),
									LOW:= REAL_TO_INT(wUsedWaterLevelOK)
									 );

				IF hsCheckUsedWaterLvl.OUT THEN
					xV_WaterOut:= 		TRUE;
					xV_UsedWaterOut:= 	FALSE;
					tnCheckWay(IN:=(*xV_WaterOutOn AND xV_NotshortcutOn AND xVoutOn*)TRUE, pt:=t#5s);
				ELSE
					xV_UsedWaterOut:= 	TRUE;
					xV_WaterOut:= 		FALSE;
					tnCheckWay(IN:=(*xV_UsedWaterOutOn AND xV_NotshortcutOn AND xVoutOn*)TRUE, pt:=t#5s);
				END_IF

				(*tnCheckWay(IN:=xV_WaterOutOn AND xV_NotshortcutOn AND xVoutOn, pt:=t#5s);*)

				*)

				IF tnCheckWay.Q THEN
					rFlawOutSet:= rFlawWaterSet;
					xPump:= 		TRUE;
				END_IF

				IF xPumpOn  THEN
					xHeaterPower:=		0;
					rToutSet:=				rTwaterSet;

				END_IF

				IF xFeedbackSwitch THEN
					xStartTimeOper:= 		TRUE;
				END_IF


				tnTimeOperation(IN:=xStartTimeOper, pt:= (WORD_TO_TIME(wRecipeTimeRinse * 1000)) - PauseOperationTime);
				wTimePassed:=REAL_TO_WORD(TIME_TO_REAL(tnTimeOperation.ET)/1000) + wTimeBeforePause;
				wTimeOperationSet:=wRecipeTimeRinse;

				IF tnTimeOperation.Q THEN
					tnTimeOperation(IN:=FALSE);
					PauseOperationTime:=T#0S;
					xStartTimeOper:= FALSE;
					State:=FindNextOperation;
				END_IF


			AlkaliIn:

				xAccidIsGoing:=		FALSE;
				xV_AlkaliOut:= 		TRUE;
				xV_AccidOut:= 		FALSE;
				xV_UsedWaterOut:= 	FALSE;
				xV_WaterOut:= 		FALSE;
				xV_Notshortcut:=		TRUE;
				xVout:= 				TRUE;

				tnCheckWay(IN:=xV_AlkaliOutOn AND xV_NotshortcutOn AND xVoutOn, pt:=t#5s);
				IF tnCheckWay.Q THEN
					rFlawOutSet:= rFlawAlcaliSet;
					xPump:= TRUE;
					State:=AlkaliInPushing;
				END_IF


			AlkaliInPushing:


				xV_AlkaliOut:= 		TRUE;
				xV_Notshortcut:=		TRUE;
				xVout:= 				TRUE;
				xPump:= 				TRUE;

				rToutSet:=				rTalcaliSet;
				rFlawOutSet:= 		rFlawAlcaliSet;

				tnCheckConc(IN:= rConcentration > rConcAlcaliSet, PT:= T#5s);
				IF tnCheckConc.Q THEN
					State:=AlkaliInWashing;
				END_IF


			AlkaliInWashing:


				xV_AlkaliOut:= 		TRUE;
				xV_Notshortcut:=		TRUE;
				xVout:= 				TRUE;
				xPump:= 				TRUE;
				xV_AlkaliIn:=			TRUE;
				(*
				xV_Cycle:=				TRUE;
				*)
				xV_Drainage:=		TRUE;
				xV_AlkaliOut:= 		TRUE;
				xV_Cycle:=			FALSE;

				rToutSet:=				rTalcaliSet;
				rFlawOutSet:= 		rFlawAlcaliSet;

				tnTimeOperation(IN:=TRUE, pt:= (WORD_TO_TIME(wRecipeTimeAlcali * 1000)) - PauseOperationTime);
				wTimePassed:=REAL_TO_WORD(TIME_TO_REAL(tnTimeOperation.ET)/1000) + wTimeBeforePause;
				wTimeOperationSet:=wRecipeTimeAlcali;

				IF tnTimeOperation.Q THEN
					tnTimeOperation(IN:=FALSE);
					PauseOperationTime:=T#0S;
					State:=FindNextOperation;
				END_IF


			WaterAfterAlkalin:


				xV_AlkaliOut:= 		FALSE;
				xV_AccidOut:= 		FALSE;
				xV_Notshortcut:=		TRUE;
				xVout:= 				TRUE;
				xPump:= 				TRUE;
				xV_Cycle:=				FALSE;


				xV_WaterOut:= 		TRUE;
				xV_UsedWaterOut:= 	FALSE;

				IF xPumpOn  THEN
					(*
					xHeaterPower:=0;*)
					rToutSet:=	wTafterAlkaliWater;

					rFlawOutSet:=rFlawWaterAfterAlcaliSet;
				END_IF

				tnCheckConc(IN:= rConcentration < wAfterRinseConcAlk, PT:= T#5s);
				IF tnCheckConc.Q THEN
					xV_AlkaliIn:=	FALSE;
					xV_Drainage:=FALSE;
				END_IF
				tnWaitZeroConc(IN:= rConcentration < 0.1, PT:= T#5s);
				IF tnWaitZeroConc.Q AND xFeedbackSwitch THEN
					xStartTimeOper:=TRUE;
				END_IF

				tnTimeOperation(IN:=xStartTimeOper, pt:= (WORD_TO_TIME(wAfterAlkWaterTime * 1000)) - PauseOperationTime);
				wTimePassed:=REAL_TO_WORD(TIME_TO_REAL(tnTimeOperation.ET)/1000) + wTimeBeforePause;
				wTimeOperationSet:=wAfterAlkWaterTime;

				IF tnTimeOperation.Q THEN
					tnTimeOperation(IN:=FALSE);
					PauseOperationTime:=T#0S;
					xStartTimeOper:=FALSE;
					State:=FindNextOperation;
				END_IF


			Accid:

				xAccidIsGoing:=		TRUE;
				xV_AccidOut:= 		TRUE;
				xV_AlkaliOut:= 		FALSE;
				xV_UsedWaterOut:= 	FALSE;
				xV_WaterOut:= 		FALSE;
				xV_Notshortcut:=		TRUE;
				xVout:= 				TRUE;

				tnCheckWay(IN:=xV_AccidOutOn AND xV_NotshortcutOn AND xVoutOn, pt:=t#5s);
				IF tnCheckWay.Q THEN
					rFlawOutSet:= rFlawAccidSet;
					xPump:= TRUE;
					State:=AccidPushing;
				END_IF


			AccidPushing:


				xV_Notshortcut:=		TRUE;
				xVout:= 				TRUE;
				xPump:= 				TRUE;
				xAccidIsGoing:=		TRUE;
				xV_AccidOut:= 		TRUE;

				rToutSet:=				rTaccidSet;
				rFlawOutSet:= 		rFlawAccidSet;

				tnCheckConc(IN:= rConcentration > rConcAccidSet, PT:= T#5s);
				IF tnCheckConc.Q THEN
					State:=AccidWashing;
				END_IF


			AccidWashing:


				xV_AccidIn:=		TRUE;
				xV_Drainage:=TRUE;
				xV_AccidOut:= TRUE;
				xV_Notshortcut:=		TRUE;
				xVout:= 				TRUE;
				xPump:= 				TRUE;

				rToutSet:=	rTaccidSet;
				rFlawOutSet:= rFlawAccidSet;

				tnTimeOperation(IN:=TRUE, pt:= (WORD_TO_TIME(wRecipeTimeAccid * 1000)) - PauseOperationTime);
				wTimePassed:=REAL_TO_WORD(TIME_TO_REAL(tnTimeOperation.ET)/1000) + wTimeBeforePause;
				wTimeOperationSet:=wRecipeTimeAccid;

				IF tnTimeOperation.Q THEN
					tnTimeOperation(IN:=FALSE);
					PauseOperationTime:=T#0S;
					State:=FindNextOperation;
				END_IF


			WaterAfterAccid:


				xV_AlkaliOut:= 		FALSE;
				xV_AccidOut:= 		FALSE;
				xV_Notshortcut:=		TRUE;
				xVout:= 				TRUE;
				xV_Cycle:=				FALSE;
				xV_WaterOut:= 		TRUE;
				xV_UsedWaterOut:= 	FALSE;
				xPump:= 				TRUE;

				IF xPumpOn  THEN
					(*
					xHeaterPower:=0;*)
					rToutSet:=	wTafterAccidWater;

					rFlawOutSet:=rFlawWaterAfterAccidSet;
				END_IF

				tnCheckConc(IN:= rConcentration <wAfterRinseConcAcc, PT:= T#5s);
				IF tnCheckConc.Q THEN
					xV_AccidIn:=		FALSE;
					xV_Drainage:=FALSE;
				END_IF
				tnWaitZeroConc(IN:= rConcentration < 0.1, PT:= T#5s);
				IF tnWaitZeroConc.Q AND xFeedbackSwitch THEN
					xStartTimeOper:=TRUE;
				END_IF
				(*
				IF NOT xV_AccidIn  THEN
					IF arOperations3x[wLine,wChosenRecipeLine ,6] THEN
						xV_Drainage:=FALSE;
					ELSE
						hsCheckUsedWaterLvl(
										IN:=(REAL_TO_INT(rUsedWaterLevel)),
										HIGH:= ( REAL_TO_INT(99)),
										LOW:= (REAL_TO_INT(97))
										 );
	
						IF hsCheckUsedWaterLvl.OUT THEN
							xV_Drainage:=TRUE;
							xV_UsedWaterIn:=TRUE;
						ELSE
							xV_Drainage:=FALSE;
						END_IF
					END_IF
				END_IF
				*)

				xV_UsedWaterIn:=FALSE;

				tnTimeOperation(IN:=xStartTimeOper, pt:= (WORD_TO_TIME(wAfterAccWaterTime * 1000)) - PauseOperationTime);
				wTimePassed:=REAL_TO_WORD(TIME_TO_REAL(tnTimeOperation.ET)/1000) + wTimeBeforePause;
				wTimeOperationSet:=wAfterAccWaterTime;

				IF tnTimeOperation.Q THEN
					tnTimeOperation(IN:=FALSE);
					PauseOperationTime:=T#0S;
					xStartTimeOper:=FALSE;
					State:=FindNextOperation;
				END_IF


			Sterelisation:

				xV_Notshortcut:=	TRUE;
				xVout:= 			TRUE;
				xV_AlkaliOut:= 	FALSE;
				xV_AccidOut:= 	FALSE;
				xV_WaterOut:= 	TRUE;
				xV_UsedWaterIn:=FALSE;
				tnCheckWay(IN:=xV_WaterOutOn AND xV_NotshortcutOn AND xVoutOn, pt:=t#5s);
				IF tnCheckWay.Q THEN
					rFlawOutSet:= wFlawSteril;
					xPump:= TRUE;
					IF wTsteril > 98 THEN
						State:= HotWaterSterilisation;
					ELSE
						xPA:=TRUE;
						xCheckConc:=TRUE;
						State:= SolutionSterilisation;
					END_IF
				END_IF


			HotWaterSterilisation:


				xV_Cycle:=			TRUE;
				xV_Drainage:=	TRUE;
				xV_Notshortcut:=		TRUE;
				xVout:= 				TRUE;
				xPump:= 				TRUE;

				xV_UsedWaterIn:=FALSE;

				rFlawOutSet:= wFlawSteril;

				IF xPumpOn  THEN
					xHeaterPower:=0;
					rToutSet:=	99;
				END_IF

				tnCheckConc(IN:= wBackTget > 85, PT:= T#5s);
				IF tnCheckConc.Q THEN
					xV_WaterOut:=	 FALSE;
					xStartTimeOper:=	TRUE;
				END_IF

				tnTimeOperation(IN:=xStartTimeOper, pt:= (WORD_TO_TIME(wSterilTime * 1000)) - PauseOperationTime);
				wTimePassed:=REAL_TO_WORD(TIME_TO_REAL(tnTimeOperation.ET)/1000) + wTimeBeforePause;
				wTimeOperationSet:=wSterilTime;

				IF tnTimeOperation.Q THEN
					tnTimeOperation(IN:=FALSE);
					PauseOperationTime:=T#0S;
					xStartTimeOper:= FALSE;
					State:=FindNextOperation;
				END_IF


			SolutionSterilisation:


				xV_Cycle:=			TRUE;
				xV_Drainage:=	TRUE;

				xV_Notshortcut:=	TRUE;
				xVout:= 			TRUE;
				xPump:= 			TRUE;
				xV_UsedWaterIn:=FALSE;

				rFlawOutSet:= wFlawSteril;
				rToutSet:= wTsteril;

				tnSolutionPortion(IN:=xPA, PT:= (WORD_TO_TIME(wConcPumpTime)*1000));
				IF tnSolutionPortion.Q THEN
					xPA:=FALSE;
					xV_WaterOut:=	FALSE;
					xStartTimeOper:=	TRUE;
					tnSolutionPortion(IN:=xPA);
				END_IF
				(*
				tnCheckConc(IN:=TRUE, PT:=(WORD_TO_TIME(wConcMessureTime)*1000));
				IF tnCheckConc.Q THEN
					tnCheckConc(IN:=FALSE);
					IF rConcentration < rConcSteril THEN
						xPA:=TRUE;
					END_IF
				END_IF
				
				IF tnCheckConc.Q AND (NOT xStartTimeOper) THEN
					xStartTimeOper:=	TRUE;
				END_IF
				

				tnWaitConc(IN:= rConcentration > rConcSteril, PT:= T#5s);
				IF tnCheckConc.Q AND (NOT xStartTimeOper) THEN
					xStartTimeOper:=	TRUE;
				END_IF
				*)

				tnTimeOperation(IN:=xStartTimeOper, pt:= (WORD_TO_TIME(wSterilTime * 1000)) - PauseOperationTime);
				wTimePassed:=REAL_TO_WORD(TIME_TO_REAL(tnTimeOperation.ET)/1000) + wTimeBeforePause;
				wTimeOperationSet:=wSterilTime;

				IF tnTimeOperation.Q THEN
					tnTimeOperation(IN:=FALSE);
					xPA:=				FALSE;
					PauseOperationTime:=T#0S;
					xStartTimeOper:= FALSE;
					State:=FindNextOperation;
				END_IF



			WaterAfterSterilisation:

				xV_AlkaliOut:= 		FALSE;
				xV_AccidOut:= 		FALSE;
				xV_Cycle:=				FALSE;
				xPA:=					FALSE;
				xV_WaterOut:= 		TRUE;
				xV_UsedWaterOut:= 	FALSE;

				xV_Notshortcut:=		TRUE;
				xVout:= 				TRUE;
				xPump:= 				TRUE;
				xV_Drainage:=		FALSE;

				IF xPumpOn  THEN
					(*
					xHeaterPower:=0;*)
					rToutSet:=	rWaterAfterSterilT;
					
					rFlawOutSet:=rWaterAfterSterilFlaw;
				END_IF

				tnCheckConc(IN:= TRUE, PT:= T#5s);
				IF tnCheckConc.Q THEN
					tnCheckConc(IN:= FALSE);
					xStartTimeOper:=TRUE;
				END_IF

				(*
				hsCheckUsedWaterLvl(
									IN:=(REAL_TO_INT(rUsedWaterLevel)),
									HIGH:= ( REAL_TO_INT(99)),
									LOW:= (REAL_TO_INT(97))
									 );

				IF hsCheckUsedWaterLvl.OUT THEN
					xV_Drainage:=TRUE;
					xV_UsedWaterIn:=TRUE;
				ELSE
					xV_Drainage:=FALSE;
					xV_UsedWaterIn:=FALSE;
				END_IF
				*)

				tnTimeOperation(IN:=xStartTimeOper, pt:= (WORD_TO_TIME(rWaterAfterSterilTime * 1000)) - PauseOperationTime);
				wTimePassed:=REAL_TO_WORD(TIME_TO_REAL(tnTimeOperation.ET)/1000) + wTimeBeforePause;
				wTimeOperationSet:=rWaterAfterSterilTime;

				IF tnTimeOperation.Q THEN
					tnTimeOperation(IN:=FALSE);
					PauseOperationTime:=T#0S;
					xStartTimeOper:=FALSE;
					State:=FindNextOperation;
				END_IF




END_CASE




tnNoFlawErr(IN:= (NOT xFeedbackSwitch) AND State > 0 AND State < 16 AND (NOT xResetErrors), PT:=t#180S);
rtErrNoFlaw(CLK:=tnNoFlawErr.Q);
IF rtErrNoFlaw.Q THEN
	xPause:=TRUE;
	wError.1:=TRUE;
END_IF

rtPumpAlm(CLK:=State > 0 AND State < 16 AND (NOT xPumpNorm));
IF rtPumpAlm.Q THEN
	xPause:=TRUE;
	wError.0:=TRUE;
END_IF

IF xResetErrors THEN


	wError:=0;
END_IF
(*
IF NOT xStartTimeOper THEN
	PauseOperationTime:=T#0S;
END_IF
*)
END_FUNCTION_BLOCK

(* POU Device/AI_Conversion/prValue_to_AO, ST *)
PROGRAM prValue_to_AO
VAR
	PumpOut_1: LIN_TRAFO;
	PumpOut_2: LIN_TRAFO;
	PumpOut_3: LIN_TRAFO;
	PumpOut_4: LIN_TRAFO;

	HeaterOut_1: LIN_TRAFO;
	HeaterOut_2: LIN_TRAFO;
	HeaterOut_3: LIN_TRAFO;
	HeaterOut_4: LIN_TRAFO;
END_VAR
PumpOut_1(
	IN:= PumpSpeedSet_1,
	IN_MIN:= 0,
	IN_MAX:= 50,
	OUT_MIN:= 0,
	OUT_MAX:= 32762,
	ERROR=> );
	AO_PumpSpeedSet_1:= REAL_TO_WORD(PumpOut_1.OUT);

PumpOut_2(
	IN:= PumpSpeedSet_2,
	IN_MIN:= 0,
	IN_MAX:= 50,
	OUT_MIN:= 0,
	OUT_MAX:= 32762,
	ERROR=> );
	AO_PumpSpeedSet_2:= REAL_TO_WORD(PumpOut_2.OUT);

PumpOut_3(
	IN:= PumpSpeedSet_3,
	IN_MIN:= 0,
	IN_MAX:= 50,
	OUT_MIN:= 0,
	OUT_MAX:= 32762,
	ERROR=> );
	AO_PumpSpeedSet_3:= REAL_TO_WORD(PumpOut_3.OUT);

PumpOut_4(
	IN:= PumpSpeedSet_4,
	IN_MIN:= 0,
	IN_MAX:= 50,
	OUT_MIN:= 0,
	OUT_MAX:= 32762,
	ERROR=> );
	AO_PumpSpeedSet_4:= REAL_TO_WORD(PumpOut_4.OUT);


HeaterOut_1(
	IN:= HeaterPowerSet_1,
	IN_MIN:= 0,
	IN_MAX:= 100,
	OUT_MIN:= 0,
	OUT_MAX:= 32762,
	ERROR=> );
	AO_HeaterPowerSet_1:= REAL_TO_WORD(HeaterOut_1.OUT);

HeaterOut_2(
	IN:= HeaterPowerSet_2,
	IN_MIN:= 0,
	IN_MAX:= 100,
	OUT_MIN:= 0,
	OUT_MAX:= 32762,
	ERROR=> );
	AO_HeaterPowerSet_2:= REAL_TO_WORD(HeaterOut_2.OUT);


HeaterOut_3(
	IN:= HeaterPowerSet_3,
	IN_MIN:= 0,
	IN_MAX:= 100,
	OUT_MIN:= 0,
	OUT_MAX:= 32762,
	ERROR=> );
	AO_HeaterPowerSet_3:= REAL_TO_WORD(HeaterOut_3.OUT);

HeaterOut_4(
	IN:= HeaterPowerSet_4,
	IN_MIN:= 0,
	IN_MAX:= 100,
	OUT_MIN:= 0,
	OUT_MAX:= 32762,
	ERROR=> );
	AO_HeaterPowerSet_4:= REAL_TO_WORD(HeaterOut_4.OUT);
END_PROGRAM

(* POU VarsToOut, ST *)
PROGRAM VarsToOut
VAR

END_VAR
_DO_PumpOn_1:= DO_PumpOn_1;
_DO_PumpOn_2:= DO_PumpOn_2;
_DO_PumpOn_3:= DO_PumpOn_3;
_DO_PumpOn_4:= DO_PumpOn_4;
 
_DO_PA11:= DO_PA11;
_DO_PA12:= DO_PA12;
_DO_PA1:= DO_PA1;
_DO_PA2:= DO_PA2;
_DO_PA3:= DO_PA3;
_DO_PA4:= DO_PA4;
 
_DO_V110:= DO_V110;
_DO_V210:= DO_V210;
_DO_V310:= DO_V310;
_DO_V410:= DO_V410;
_DO_V111:= DO_V111;
_DO_V211:= DO_V211;
_DO_V311:= DO_V311;
_DO_V411:= DO_V411;

_DO_V101:= DO_V101;
_DO_V102:= DO_V102;
_DO_V103:= DO_V103;
_DO_V104:= DO_V104;
_DO_V105:= DO_V105;
_DO_V106:= DO_V106;
_DO_V107:= DO_V107;
_DO_V108:= DO_V108;
_DO_V109:= DO_V109;
_DO_V201:= DO_V201;
_DO_V202:= DO_V202;
_DO_V203:= DO_V203;
_DO_V204:= DO_V204;
_DO_V205:= DO_V205;
_DO_V206:= DO_V206;
_DO_V207:= DO_V207;
_DO_V208:= DO_V208;
_DO_V209:= DO_V209;
_DO_V301:= DO_V301;
_DO_V302:= DO_V302;
_DO_V303:= DO_V303;
_DO_V304:= DO_V304;
_DO_V305:= DO_V305;
_DO_V306:= DO_V306;
_DO_V307:= DO_V307;
_DO_V308:= DO_V308;
_DO_V309:= DO_V309;
_DO_V401:= DO_V401;
_DO_V402:= DO_V402;
_DO_V403:= DO_V403;
_DO_V404:= DO_V404;
_DO_V405:= DO_V405;
_DO_V406:= DO_V406;
_DO_V407:= DO_V407;
_DO_V408:= DO_V408;
_DO_V409:= DO_V409;
 
_DO_V501:= DO_V501;

_DO_V511:= DO_V511;
_DO_V510:= DO_V510;
_DO_V512:= DO_V512;
_DO_V513:= DO_V513;
_DO_V514:= DO_V514;
_DO_V515:= DO_V515;


_SwitchOnRemotePump_1	:=	SwitchOnRemotePump_1	;
_SwitchOnRemotePump_2	:=	SwitchOnRemotePump_2	;
_SwitchOnRemotePump_3	:=	SwitchOnRemotePump_3	;
_SwitchOnRemotePump_4	:=	SwitchOnRemotePump_4	;


_Ready_Line_2 :=SwitchOnRemotePump_1_2;
_Working_Line_2 :=SwitchOnRemotePump_1_1;
_Working_Pump_2:=SwitchOnRemotePump_1_3;


_AO_PumpSpeedSet_1:= AO_PumpSpeedSet_1;
_AO_PumpSpeedSet_2:= AO_PumpSpeedSet_2;
_AO_PumpSpeedSet_3:= AO_PumpSpeedSet_3;
_AO_PumpSpeedSet_4:= AO_PumpSpeedSet_4;
 
_AO_HeaterPowerSet_1:= AO_HeaterPowerSet_1;
_AO_HeaterPowerSet_2:= AO_HeaterPowerSet_2;
_AO_HeaterPowerSet_3:= AO_HeaterPowerSet_3;
_AO_HeaterPowerSet_4:= AO_HeaterPowerSet_4;
END_PROGRAM

(* POU Device/AI_Conversion/prAI_to_Value, ST *)
PROGRAM prAI_to_Value
VAR
	fbCleanWaterLeve: LIN_TRAFO;
	fbUsedWaterLeve: LIN_TRAFO;
	fbAccidLevel: LIN_TRAFO;
	fbAlkaliLevel: LIN_TRAFO;

END_VAR
(*
Conc_Line1:=(AI_Conc_Line1/32765)*100;

Conc_Line2:=(AI_Conc_Line2/32765)*100;

Conc_Line3:=(AI_Conc_Line3/32765)*100;

Conc_Line4:=(AI_Conc_Line4/32765)*100;

CleanWaterLevel:=(AI_CleanWaterLevel/32765)*100;

UsedWaterLevel:=(AI_UsedWaterLevel/32765)*100;

AccidLevel:=(AI_AccidLevel/32765)*100;

AlkaliLevel:=(AI_AlkaliLevel/32765)*100;
*)
fbCleanWaterLeve(
	IN:= AI_CleanWaterLevel,
	IN_MIN:= 0,
	IN_MAX:= 32762,
	OUT_MIN:= 0,
	OUT_MAX:= 40000,
	ERROR=> );
	CleanWaterLevel:= fbCleanWaterLeve.OUT;

fbUsedWaterLeve(
	IN:= AI_UsedWaterLevel,
	IN_MIN:= 0,
	IN_MAX:= 32762,
	OUT_MIN:= 0,
	OUT_MAX:= 40000,
	ERROR=> );
	UsedWaterLevel:= fbUsedWaterLeve.OUT;

fbAccidLevel(
	IN:= AI_AccidLevel,
	IN_MIN:= 0,
	IN_MAX:= 32762,
	OUT_MIN:= 0,
	OUT_MAX:= 40000,
	ERROR=> );
	AccidLevel:= fbAccidLevel.OUT;

fbAlkaliLevel(
	IN:= AlkaliLevel,
	IN_MIN:= 0,
	IN_MAX:= 32762,
	OUT_MIN:= 0,
	OUT_MAX:= 40000,
	ERROR=> );
	AlkaliLevel:= fbAlkaliLevel.OUT;
END_PROGRAM

(* POU Process/Washing/prRemoteEquipment, ST *)
PROGRAM prRemoteEquipment
VAR
	rtRecipe_1:	R_TRIG;
	rtRecipe_2:	R_TRIG;
	rtRecipe_3:	R_TRIG;
	rtRecipe_4:	R_TRIG;
	rtRecipe_5:	R_TRIG;

	ftRecipe_1:	F_TRIG;
	ftRecipe_2:	F_TRIG;
	ftRecipe_3:	F_TRIG;
	ftRecipe_4:	F_TRIG;
	ftRecipe_5:	F_TRIG;

	xCheck: BOOL;
	xCheck1: WORD;
	tnPause:	TON;
	rtPause:R_TRIG;
END_VAR
_Ready_Line_1:= wDissolvingStateLine4 = 0 AND SelfWashState = 0 AND wWashingErr =0;
_Working_Line_1:= wWashingStateLine4>0;
_Working_Pump_1:= Pump_FeedbackOn_4;


rtRecipe_1(CLK:=Permition_Line_1);
rtRecipe_2(CLK:=Permition_Line_2);
rtRecipe_3(CLK:=Permition_Line_3);
rtRecipe_4(CLK:=Permition_Line_4);
rtRecipe_5(CLK:=Permition_Line_5);

ftRecipe_1(CLK:=Permition_Line_1 OR Permition_Line_2 OR Permition_Line_3 OR Permition_Line_4 OR Permition_Line_5);
ftRecipe_2(CLK:=Permition_Line_2);
ftRecipe_3(CLK:=Permition_Line_3);
ftRecipe_4(CLK:=Permition_Line_4);
ftRecipe_5(CLK:=Permition_Line_5);

IF rtRecipe_1.Q AND wWashingStateLine4 = 0 THEN
	wChosenRecipeLine4:=1;
	xStartWashingLine4:=TRUE;
END_IF
IF rtRecipe_2.Q AND wWashingStateLine4 = 0 THEN
	wChosenRecipeLine4:=2;
	xStartWashingLine4:=TRUE;
END_IF
IF rtRecipe_3.Q AND wWashingStateLine4 = 0 THEN
	wChosenRecipeLine4:=3;
	xStartWashingLine4:=TRUE;
END_IF
IF rtRecipe_4.Q  AND wWashingStateLine4 = 0 THEN
	wChosenRecipeLine4:=4;
	xStartWashingLine4:=TRUE;
END_IF
IF rtRecipe_5.Q AND wWashingStateLine4 = 0 THEN
	wChosenRecipeLine4:=5;
	xStartWashingLine4:=TRUE;
END_IF

IF ftRecipe_1.Q THEN
	xCheck:=TRUE;
	xCheck1:=xCheck1 + 1;
	(*xPauseWashingLine4:=TRUE;;*)
END_IF

IF Permition_Line_1 OR Permition_Line_2 OR Permition_Line_3 OR Permition_Line_4 OR Permition_Line_5 THEN
	xCheck:=FALSE;
END_IF

tnPause(IN:=xCheck, PT:= T#3S);
rtPause(CLK:=tnPause.Q);

IF rtPause.Q THEN
	xPauseWashingLine4:=TRUE;
END_IF
END_PROGRAM

(* POU Process/SelfWashing/prSelfWashing, ST *)
PROGRAM prSelfWashing
VAR
	SelfWashing:	fbSelfWashing;
	xResetErrors:	BOOL;
END_VAR
IF wWashingStateLine1 = 0 AND wDissolvingStateLine1 = 0 THEN

SelfWashing(
	rWaterLevel:= CleanWaterLevel,
	rUsedWaterLevel:= UsedWaterLevel,
	rAccidLevel:= AccidLevel,
	rAlkaliLevel:= AlkaliLevel,
	wUsedWaterLevelOK:= SelfWashUsedWaterLevelOK,
	wWaterLevelOK:= SelfWashWaterLevelOK,
	wUsedWaterLevelDrain:= SelfWashUsedWaterLevelDrain,
	wWaterLevelDrain:= SelfWashWaterLevelDrain,
	wAlkaliLevelOK:= SelfWashAlkaliLevelOK,
	wAlkaliLevelDrain:= SelfWashAlkaliLevelDrain,
	wAccidLevelOK:= SelfWashAccidLevelOK,
	wAccidLevelDrain:= SelfWashwAccidLevelDrain,
	wPumpFlawSet:= SelfWashwPumpFlawSet,
	wWashByAlkaliTime:= SelfWashByAlkaliTime,
	wWashByAccidTime:= SelfWashByAccidTime,
	wWashByWaterTime:= SelfWashByWaterTime_,
	xAlkaliCooked:= xAlkaliIsReady,
	xAccidCooked:= xAccidIsReady,
	xPause:=xSelsWashingPause,
	xVoutOn:= xState_V111,
	xV_NotshortcutOn:= xState_V110,
	xV_UsedWaterInOn:= xState_V514,
	xV_WaterInOn:= xState_V513,
	xV_UsedWaterInFillOn:= xState_V108,
	xV_AlkaliInOn:= xState_V512,
	xV_AccidInOn:= xState_V511,
	xV_WaterOutOn:= xState_V101,
	xV_UsedWaterOutOn:= xState_V102,
	xV_AlkaliOutOn:= xState_V104,
	xV_AccidOutOn:= xState_V103,
	xV_CycleOn:= xState_V105,
	xPumpOn:= Pump_OnAuto_1,
	xV_AllInOn:= xState_V510,
	xV_DrainageOn:= xState_V109,
	xDrainOk:= xDrainOk,
	Dissolving_StateLine1:= wDissolvingStateLine1,
	Dissolving_StateLine2:= wDissolvingStateLine2,
	Dissolving_StateLine3:= wDissolvingStateLine3,
	Dissolving_StateLine4:= wDissolvingStateLine4,
	xStart:= xStartSelfWashing,
	xDoWaterTank:= SelfWashDoWaterTank,
	xDoUsedWaterTank:= SelfWashDoUsedWaterTank,
	xDoAlkaliTank:= SelfWashDoAlkaliTank,
	xDoAccidTank:= SelfWashDoAccidTank,
	xVout:= OnAuto_V111,
	xV_Notshortcut:= OnAuto_V110,
	xV_WaterOut:= OnAuto_V101,
	xV_UsedWaterOut:= OnAuto_V102,
	xV_Cycle:= OnAuto_V105,
	xV_Drainage:=  OnAuto_V109,
	xV_Drainage_1:= OnAuto_V515,
	xV_AlkaliOut:= OnAuto_V104,
	xV_AccidOut:= OnAuto_V103,
	xV_WaterIn:= OnAuto_V513,
	xV_UsedWaterIn:= OnAuto_V514,
	xV_UsedWaterInFill:= OnAuto_V108,
	xV_AlkaliIn:= OnAuto_V512,
	xV_AccidIn:= OnAuto_V511,
	xV_AllIn:= OnAuto_V510,
	xPump:= Pump_OnAuto_1,
	xResetErrors:= xResetErrors,
	xAcknawlage:=SelfWashingAcknawlage,
	wPumpFlawOut:= (*WORD_TO_REAL(Pump_FlawManualSet_1)*)SelfWashwPumpFlawSet,
	xDoDissolveAlkali:= xDissolDoAlkali,
	xDoDissolveAccid:= xDissilDoAccid,
	xStartDissolving:= xDissolving_Start,
	xV_UsedWaterInFill:=OnAuto_V108,
	xStopFillingWaterTank:= xStopFillingWaterTank,
	rFlawSet:= Pump_FlawAutoSet_1,
	State=> SelfWashState,
	PauseState=> SelfWashPauseState,
	wError=> ,
	xWaterIsReady=> SelfWashWaterIsReady,
	xUsedWaterIsReady=> SelfWashUsedWaterIsReady,
	xAlkaliIsReady=> SelfWashAlkaliIsReady,
	wTimePassed=> SelfWashingTimePast,
	wTimeOperationSet=> SelfWashingOperTimeSet,
	xAccidIsReady=> SelfWashAccidIsReady);

END_IF

prSelfWashStateBits();
END_PROGRAM

(* POU Process/SelfWashing/fbSelfWashing, ST *)
FUNCTION_BLOCK fbSelfWashing
VAR_INPUT

	rWaterLevel:					REAL;
	rUsedWaterLevel:				REAL;
	rAccidLevel:					REAL;
	rAlkaliLevel:					REAL;
	wUsedWaterLevelOK: 		REAL;
	wWaterLevelOK: 				REAL;
	wUsedWaterLevelDrain: 		REAL;
	wWaterLevelDrain: 			REAL;
	wAlkaliLevelOK: 				REAL;
	wAlkaliLevelDrain: 			REAL;
	wAccidLevelOK: 				REAL;
	wAccidLevelDrain: 			REAL;
	wPumpFlawSet:				REAL;
	wWashByAlkaliTime:			WORD;
	wWashByAccidTime:			WORD;
	wWashByWaterTime:			WORD;

	xAlkaliCooked:				BOOL;
	xAccidCooked:				BOOL;

	xVoutOn:						BOOL;
	xV_NotshortcutOn:			BOOL;
	xV_UsedWaterInOn:			BOOL;
	xV_WaterInOn:			BOOL;
	xV_UsedWaterInFillOn:		BOOL;
	xV_AlkaliInOn:					BOOL;
	xV_AccidInOn:					BOOL;
	xV_WaterOutOn:				BOOL;
	xV_UsedWaterOutOn:			BOOL;
	xV_AlkaliOutOn:				BOOL;
	xV_AccidOutOn:				BOOL;
	xV_CycleOn:					BOOL;
	xPumpOn:						BOOL;
	xV_AllInOn:					BOOL;
	xV_DrainageOn:				BOOL;
	xPause:						BOOL;


	Dissolving_StateLine1:				Dissolving_States;
	Dissolving_StateLine2:				Dissolving_States;
	Dissolving_StateLine3:				Dissolving_States;
	Dissolving_StateLine4:				Dissolving_States;
	wPumpFlawOut:			REAL;

END_VAR
VAR_IN_OUT

	xStart:						BOOL;

	xDrainOk:						BOOL;

	xDoWaterTank:				BOOL;
	xDoUsedWaterTank:			BOOL;
	xDoAlkaliTank:					BOOL;
	xDoAccidTank:					BOOL;

	xVout:						BOOL;
	xV_Notshortcut:			BOOL;
	xV_WaterOut:				BOOL;
	xV_UsedWaterOut:		BOOL;
	xV_Cycle:					BOOL;
	xV_Drainage:				BOOL;
	xV_Drainage_1:			BOOL;
	xV_AlkaliOut:				BOOL;
	xV_AccidOut:				BOOL;
	xV_WaterIn:				BOOL;
	xV_UsedWaterIn:			BOOL;
	xV_UsedWaterInFill:			BOOL;
	xV_AlkaliIn:				BOOL;
	xV_AccidIn:				BOOL;
	xV_AllIn:					BOOL;


	xPump:					BOOL;
	xResetErrors:				BOOL;

	xDoDissolveAlkali:		BOOL;
	xDoDissolveAccid:		BOOL;
	xStartDissolving:			BOOL;
	xStopFillingWaterTank:	BOOL;
	xAcknawlage:				BOOL;
	rFlawSet:					REAL;


END_VAR
VAR_OUTPUT
	State:						SelfWashingStates;
	PauseState:				SelfWashingStates;
	wError:						WORD;
	xWaterIsReady:			BOOL;
	xUsedWaterIsReady:		BOOL;
	xAlkaliIsReady:			BOOL;
	xAccidIsReady:			BOOL;
	wTimePassed:			WORD;
	wTimeOperationSet:		WORD;
END_VAR
VAR
	rtStart:					R_TRIG;
	rtPause:				R_TRIG;
	ftStart:					F_TRIG;
	tnWashing:			TON;
	xStartOper:			BOOL;
	xDissolvingStoped:	BOOL;
	xWaterCleaned:		BOOL;
	xUsedWaterCleaned:	BOOL;
	xAlkaliCleaned:		BOOL;
	XAccidCleaned:		BOOL;
	PauseOperationTime:	TIME;
	wTimeBeforePause:			WORD;
	wNextState:			SelfWashingStates;
	xUsedWaterAlkaliClined:	BOOL;
	xCleanWaterAlkaliClined:	BOOL;
END_VAR
rtStart(CLK:=xStart);
ftStart(CLK:=xStart);
rtPause(CLK:=xPause);

IF rtStart.Q THEN
	xVout:=						FALSE;
	xV_Notshortcut:=			FALSE;
	xAlkaliIsReady:=			NOT xDoAlkaliTank;
	xAccidIsReady:=			NOT xDoAccidTank;
	xWaterIsReady:=			NOT xDoWaterTank;
	xUsedWaterIsReady:=	NOT xDoUsedWaterTank;
	rFlawSet:=					wPumpFlawSet;

	IF (NOT(xDoUsedWaterTank OR xDoWaterTank OR xDoAccidTank)) AND xDoAlkaliTank THEN
		wNextState:=WashAlkaliTankWater;
		State:= EmptyAlkaliTank;
	ELSIF (NOT(xDoUsedWaterTank OR xDoWaterTank OR xDoAlkaliTank)) AND xDoAccidTank THEN
		wNextState:=WashAccidTankWater;
		State:=EmptyAccidTank;
	ELSIF xDoUsedWaterTank OR xDoWaterTank  THEN
		wNextState:=CheckAll;
		State:=EmptyUsedWaterTank;
	ELSE
		State:=CheckAll;
	END_IF

END_IF

IF ftStart.Q THEN
	wError:=0;
	xVout:=						FALSE;
	xV_Notshortcut:=			FALSE;
	xV_WaterOut:=			FALSE;
	xV_Cycle:=					FALSE;
	xV_Drainage:=			FALSE;
	xV_AlkaliOut:=				FALSE;
	xV_AccidOut:=				FALSE;
	xV_AlkaliIn:=				FALSE;
	xV_AccidIn:=				FALSE;
	xV_WaterIn:=				FALSE;
	xPump:=					FALSE;
	xStartOper:=				FALSE;
	xV_Drainage_1:=			FALSE;
	xStopFillingWaterTank:=	FALSE;
	xWaterCleaned:=			FALSE;
	xUsedWaterCleaned:=	FALSE;
	xAlkaliCleaned:=			FALSE;
	XAccidCleaned:=			FALSE;
	wTimeOperationSet:=		0;
	xV_UsedWaterIn:=		FALSE;
	xV_UsedWaterInFill:=		FALSE;
	xAcknawlage:=			FALSE;
	xV_AllIn:=					FALSE;
	wTimePassed:=			0;
	wTimeBeforePause:=		0;
	PauseOperationTime:=	T#0S;
	xV_UsedWaterOut:=		FALSE;
	xUsedWaterAlkaliClined:=FALSE;
	xCleanWaterAlkaliClined:=FALSE;
	wNextState:=			StopSelfWashing;
	State:=					StopSelfWashing;
END_IF


IF rtPause.Q THEN
	PauseState:=State;
	PauseOperationTime:=tnWashing.ET;
	wTimeBeforePause:=wTimePassed;
	PauseOperationTime:=PauseOperationTime + tnWashing.ET;
	tnWashing(IN:=FALSE);
	State:=SelfWashingPause;
END_IF

xDissolvingStoped:= Dissolving_StateLine1 = DissolvingStop AND Dissolving_StateLine2 = DissolvingStop
						AND Dissolving_StateLine3 = DissolvingStop AND Dissolving_StateLine4 = DissolvingStop;




CASE State OF


			StopSelfWashing:
								;


			SelfWashingPause:


				IF NOT xPause THEN
					State:=PauseState;
				END_IF


			CheckAll:


				IF rAlkaliLevel >= wAlkaliLevelOK  AND rAccidLevel >= wAccidLevelOK  AND xDissolvingStoped THEN
					IF xDoWaterTank OR xDoUsedWaterTank THEN
						wNextState:=WashUsedWaterTankAlkali;
						State:=WashUsedWaterTankWater;
					ELSIF xDoAlkaliTank THEN
						wNextState:=WashAlkaliTankWater;
						State:=EmptyAlkaliTank;
					ELSIF xDoAccidTank THEN
						wNextState:=WashAccidTankWater;
						State:=EmptyAccidTank;
					END_IF
				ELSE
					(*xDoDissolveAlkali:=TRUE;
					xDoDissolveAccid:= TRUE;
					xStartDissolving:=TRUE;*)
					State:= WaitAllDissolving;
					xAcknawlage:=TRUE;
				END_IF

			WaitAllDissolving:

				xV_UsedWaterOut:=		FALSE;
				xPump:=					FALSE;

				IF rAlkaliLevel >= wAlkaliLevelOK AND xAlkaliCooked
					AND  rAccidLevel >= wAccidLevelOK AND xAccidCooked  AND xDissolvingStoped AND (NOT xAcknawlage) THEN
					State:=CheckAll;
				END_IF



			EmptyUsedWaterTank:


				xVout:=					FALSE;
				xV_Notshortcut:=		FALSE;
				xV_Drainage:=		FALSE;
				xV_AllIn:=				FALSE;
				xV_Drainage_1:=		FALSE;
				xV_UsedWaterIn:=	FALSE;
				xV_WaterOut:=		FALSE;
				xV_UsedWaterOut:=	TRUE;

				IF (NOT (xVoutOn OR xV_NotshortcutOn OR xV_DrainageOn)) AND xV_UsedWaterOutOn  THEN
					xPump:=TRUE;
				END_IF

				IF rUsedWaterLevel < wUsedWaterLevelDrain THEN
					(*
					IF xUsedWaterCleaned THEN
						xUsedWaterCleaned:= FALSE;
						State:= FillUsedWaterTank;
					ELSE
						State:= CheckAll;
					END_IF
					*)
					State:= wNextState;
				END_IF


			WashUsedWaterTankAlkali:


				xV_AllIn:=				TRUE;
				xV_Drainage_1:=		TRUE;
				xV_Drainage:=		TRUE;
				xV_UsedWaterIn:=	TRUE;
				xV_AlkaliOut:=			TRUE;
				xV_UsedWaterOut:=	FALSE;
				xV_WaterOut:=		FALSE;

				IF (NOT xV_UsedWaterOutOn) AND xV_AllInOn AND xV_UsedWaterInOn AND xV_AlkaliOutOn THEN
					xPump:=TRUE;
					xStartOper:=TRUE;
				END_IF

				tnWashing(IN:=xStartOper,  PT:= ((WORD_TO_TIME(wWashByAlkaliTime))*1000) - PauseOperationTime);
				wTimePassed:=REAL_TO_WORD(TIME_TO_REAL(tnWashing.ET)/1000) + wTimeBeforePause;
				wTimeOperationSet:=wWashByAlkaliTime;

				IF tnWashing.Q THEN
					tnWashing(IN:=FALSE);
					xStartOper:=FALSE;
					wTimePassed:=		0;
					wTimeBeforePause:=0;
					PauseOperationTime:=T#0S;
					xUsedWaterAlkaliClined:=TRUE;
					wNextState:=WashUsedWaterTankWater;
					State:= EmptyUsedWaterTank;
				END_IF




			WashUsedWaterTankAccid:


				xV_AllIn:=				TRUE;
				xV_Drainage_1:=		TRUE;
				xV_Drainage:=		TRUE;
				xV_UsedWaterIn:=	TRUE;
				xV_AccidOut:=			TRUE;
				xV_AlkaliOut:=			FALSE;
				xV_UsedWaterOut:=	FALSE;
				xV_WaterOut:=		FALSE;

				IF (NOT xV_AlkaliOutOn) AND xV_AllInOn AND xV_UsedWaterInOn AND xV_AccidOutOn THEN
					xPump:=TRUE;
					xStartOper:=TRUE;
				END_IF

				tnWashing(IN:=xStartOper,  PT:= ((WORD_TO_TIME(wWashByAccidTime))*1000) - PauseOperationTime);
				wTimePassed:=REAL_TO_WORD(TIME_TO_REAL(tnWashing.ET)/1000) + wTimeBeforePause;
				wTimeOperationSet:=wWashByAccidTime;

				IF tnWashing.Q THEN
					tnWashing(IN:=FALSE);
					xStartOper:=FALSE;
					wTimePassed:=		0;
					PauseOperationTime:=T#0S;
					wTimeBeforePause:=0;
					xUsedWaterCleaned:=TRUE;
					wNextState:=WashUsedWaterTankWater;
					State:= EmptyUsedWaterTank;
				END_IF


			WashUsedWaterTankWater:


				xV_AllIn:=				TRUE;
				xV_Drainage_1:=		TRUE;
				xV_Drainage:=		TRUE;
				xV_UsedWaterIn:=	TRUE;
				xV_WaterOut:=		TRUE;
				xV_AccidOut:=			FALSE;
				xV_AlkaliOut:=				FALSE;
				xV_UsedWaterOut:=	FALSE;


				IF (NOT xV_AlkaliOutOn) AND xV_AllInOn AND xV_UsedWaterInOn  THEN
					xPump:=TRUE;
					xStartOper:=TRUE;
				END_IF

				tnWashing(IN:=xStartOper,  PT:= ((WORD_TO_TIME(wWashByWaterTime))*1000) - PauseOperationTime);
				wTimePassed:=REAL_TO_WORD(TIME_TO_REAL(tnWashing.ET)/1000) + wTimeBeforePause;
				wTimeOperationSet:=wWashByWaterTime;

				IF tnWashing.Q THEN
					tnWashing(IN:=FALSE);
					xStartOper:=FALSE;
					wTimePassed:=		0;
					PauseOperationTime:=T#0S;
					wTimeBeforePause:=0;

					IF xUsedWaterCleaned AND xUsedWaterAlkaliClined THEN
						wNextState:= FillUsedWaterTank;
					ELSIF xUsedWaterAlkaliClined THEN
						wNextState:= WashUsedWaterTankAccid;
					ELSE
						wNextState:= WashUsedWaterTankAlkali;
					END_IF
					State:=EmptyUsedWaterTank;
				END_IF



			FillUsedWaterTank:


				xV_WaterOut:=		TRUE;
				xV_UsedWaterInFill:=	TRUE;
				xV_Drainage_1:=		FALSE;
				xV_Drainage:=		TRUE;
				xV_AllIn:=				FALSE;
				xV_UsedWaterIn:=	FALSE;
				xPump:=			TRUE;
				xV_UsedWaterOut:=	FALSE;
				IF xDoWaterTank THEN
					xStopFillingWaterTank:=	TRUE;
				ELSE
					xStopFillingWaterTank:=	FALSE;
				END_IF



				IF rUsedWaterLevel > wUsedWaterLevelOK OR (NOT xDoWaterTank) THEN
					IF xDoWaterTank  THEN
						wNextState:=WashWaterTankWater;
						State:=EmptyWaterTank;
					ELSIF xDoAlkaliTank THEN
						wNextState:=WashAlkaliTankWater;
						State:=EmptyAlkaliTank;
					ELSIF xDoAccidTank THEN
						wNextState:=WashAccidTankWater;
						State:=EmptyAccidTank;
					ELSE
						xStart:=FALSE;
					END_IF
				END_IF


			EmptyWaterTank:

				xStopFillingWaterTank:=	TRUE;;
				xV_WaterOut:=			TRUE;
				xV_AlkaliOut:=				FALSE;
				xV_AccidOut:=				FALSE;
				xV_Drainage:=			FALSE;
				xV_UsedWaterIn:=		FALSE;
				xV_UsedWaterInFill:=		FALSE;

				IF (NOT xV_DrainageOn)  AND xV_WaterOutOn THEN
					xPump:=TRUE;
				END_IF

				IF rWaterLevel < wWaterLevelDrain THEN
					(*
					IF xWaterCleaned THEN
						xWaterCleaned:=FALSE;
						xStopFillingWaterTank:=	FALSE;
						State:= FillWaterTank;
					ELSE
					State:= WashWaterTankAlkali;
					END_IF
					*)
					State:=wNextState;
				END_IF



			WashWaterTankAlkali:


				xStopFillingWaterTank:=	TRUE;
				xV_AllIn:=					TRUE;
				xV_Drainage_1:=			TRUE;
				xV_Drainage:=			TRUE;
				xV_WaterIn:=				TRUE;
				xV_AlkaliOut:=				TRUE;
				xV_UsedWaterOut:=		FALSE;
				xV_WaterOut:=			FALSE;

				IF (NOT xV_UsedWaterOutOn) AND xV_AllInOn AND xV_WaterInOn AND xV_AlkaliOutOn THEN
					xPump:=TRUE;
					xStartOper:=TRUE;
				END_IF

				tnWashing(IN:=xStartOper,  PT:= ((WORD_TO_TIME(wWashByAlkaliTime))*1000) - PauseOperationTime);
				wTimePassed:=REAL_TO_WORD(TIME_TO_REAL(tnWashing.ET)/1000) + wTimeBeforePause;
				wTimeOperationSet:=wWashByAlkaliTime;

				IF tnWashing.Q THEN
					tnWashing(IN:=FALSE);
					xStartOper:=FALSE;
					wTimePassed:=		0;
					PauseOperationTime:=T#0S;
					wTimeBeforePause:=0;
					xCleanWaterAlkaliClined:=TRUE;
					wNextState:= WashWaterTankWater;
					State:= EmptyWaterTank;
				END_IF


			WashWaterTankAccid:


				xStopFillingWaterTank:=	TRUE;
				xV_AllIn:=					TRUE;
				xV_Drainage_1:=			TRUE;
				xV_Drainage:=			TRUE;
				xV_WaterIn:=				TRUE;
				xV_AccidOut:=				TRUE;
				xV_AlkaliOut:=				FALSE;
				xV_WaterOut:=			FALSE;
				xV_UsedWaterOut:=		FALSE;

				IF (NOT xV_AlkaliOutOn) AND xV_AllInOn AND xV_WaterInOn AND xV_AccidOutOn THEN
					xPump:=TRUE;
					xStartOper:=TRUE;
				END_IF

				tnWashing(IN:=xStartOper,  PT:= ((WORD_TO_TIME(wWashByAccidTime))*1000) - PauseOperationTime);
				wTimePassed:=REAL_TO_WORD(TIME_TO_REAL(tnWashing.ET)/1000) + wTimeBeforePause;
				wTimeOperationSet:=wWashByAccidTime;

				IF tnWashing.Q THEN
					tnWashing(IN:=FALSE);
					xStartOper:=FALSE;
					wTimePassed:=		0;
					PauseOperationTime:=T#0S;
					wTimeBeforePause:=0;
					xWaterCleaned:=	TRUE;
					wNextState:=WashWaterTankWater;
					State:= EmptyWaterTank;
				END_IF



			WashWaterTankWater:


				xStopFillingWaterTank:=	TRUE;
				xV_AllIn:=					TRUE;
				xV_Drainage_1:=			TRUE;
				xV_Drainage:=			TRUE;
				xV_WaterIn:=				TRUE;
				xV_UsedWaterOut:=		TRUE;
				xV_AccidOut:=				FALSE;
				xV_WaterOut:=			FALSE;
				xV_AlkaliOut:=				FALSE;
				xV_WaterOut:=			FALSE;


				IF (NOT xV_AccidOutOn) AND xV_AllInOn AND xV_WaterInOn  THEN
					xPump:=TRUE;
					xStartOper:=TRUE;
				END_IF

				tnWashing(IN:=xStartOper,  PT:= ((WORD_TO_TIME(wWashByWaterTime))*1000) - PauseOperationTime);
				wTimePassed:=REAL_TO_WORD(TIME_TO_REAL(tnWashing.ET)/1000) + wTimeBeforePause;
				wTimeOperationSet:=wWashByWaterTime;

				IF tnWashing.Q THEN
					tnWashing(IN:=FALSE);
					xStartOper:=		FALSE;
					wTimePassed:=		0;
					PauseOperationTime:=T#0S;
					wTimeBeforePause:=0;
					(*
					IF xWaterCleaned THEN
						State:= EmptyWaterTank;
					ELSE
						State:=WashWaterTankAccid;
					END_IF
					*)
					IF xWaterCleaned AND xCleanWaterAlkaliClined THEN
						wNextState:= FillUsedWaterTank;
					ELSIF xCleanWaterAlkaliClined THEN
						wNextState:= WashWaterTankAccid;
					ELSE
						wNextState:= WashWaterTankAlkali;
					END_IF
					State:= EmptyWaterTank;
				END_IF



			FillWaterTank:


				xStopFillingWaterTank:=	FALSE;
				xV_AllIn:=					FALSE;
				xV_Drainage_1:=			FALSE;
				xV_Drainage:=			FALSE;
				xV_WaterIn:=				FALSE;
				xV_WaterOut:=			FALSE;
				xV_AccidOut:=				FALSE;
				xV_UsedWaterOut:=		FALSE;
				xPump:=					TRUE;

				(*IF rWaterLevel > wWaterLevelOK THEN*)
					IF xDoAlkaliTank THEN
						wNextState:=WashAlkaliTankWater;
						State:=EmptyAlkaliTank;
					ELSIF xDoAccidTank THEN
						wNextState:=WashAccidTankWater;
						State:=EmptyAccidTank;
					ELSE
						xStart:=FALSE;
					END_IF
				(*END_IF*)



			EmptyAlkaliTank:



				xV_AlkaliOut:=				TRUE;
				xV_WaterOut:=			FALSE;
				xV_AccidOut:=				FALSE;
				xV_Drainage:=			FALSE;
				xV_UsedWaterInFill:=		FALSE;

				IF (NOT xV_DrainageOn) AND xV_AllInOn AND xV_AlkaliOutOn THEN
					xPump:=TRUE;
				END_IF

				IF rAlkaliLevel < wAlkaliLevelDrain THEN
					xPump:= FALSE;
					xAcknawlage:=TRUE;
					State:= WaitManualAlkaliDrain;
				END_IF



			WaitManualAlkaliDrain:


				xPump:= 					FALSE;
				xV_AlkaliOut:=				FALSE;
				xV_AllIn:=					FALSE;
				xV_AlkaliIn:=				FALSE;

				IF NOT  xAcknawlage THEN
						(*
						IF xAlkaliCleaned THEN
							xAlkaliCleaned:=FALSE;
							(*
							xDoDissolveAlkali:=TRUE;
							xStartDissolving:=TRUE;
							*)
							xAcknawlage:=TRUE;
							State:= FillAlkaliTank;
						ELSE
						State:= WashAlkaliTankWater;
						END_IF
						*)
					State:=wNextState;
				END_IF



			WashAlkaliTankAccid:


				xV_AllIn:=					TRUE;
				xV_Drainage_1:=			TRUE;
				xV_Drainage:=			TRUE;
				xV_AlkaliIn:=				TRUE;
				xV_AccidOut:=				TRUE;
				xV_AlkaliOut:=				FALSE;
				xV_WaterOut:=			FALSE;

				IF (NOT xV_AlkaliOutOn) AND xV_AllInOn AND xV_AlkaliInOn AND xV_AccidOutOn THEN
					xPump:=TRUE;
					xStartOper:=TRUE;
				END_IF

				tnWashing(IN:=xStartOper,  PT:= ((WORD_TO_TIME(wWashByAccidTime))*1000 - PauseOperationTime));
				wTimePassed:=REAL_TO_WORD(TIME_TO_REAL(tnWashing.ET)/1000) + wTimeBeforePause;
				wTimeOperationSet:=wWashByAccidTime;

				IF tnWashing.Q THEN
					tnWashing(IN:=FALSE);
					xStartOper:=FALSE;
					wTimePassed:=		0;
					PauseOperationTime:=T#0S;
					wTimeBeforePause:=0;
					xAlkaliCleaned:= 	TRUE;
					wNextState:=FillAlkaliTank;
					State:= WashAlkaliTankWater;
				END_IF


			WashAlkaliTankWater:


				xV_AllIn:=				TRUE;
				xV_Drainage_1:=		TRUE;
				xV_Drainage:=		TRUE;
				xV_AlkaliIn:=			TRUE;
				xV_WaterOut:=		TRUE;
				xV_AccidOut:=			FALSE;


				IF (NOT xV_AlkaliOutOn) AND xV_AllInOn AND xV_AlkaliInOn  THEN
					xPump:=TRUE;
					xStartOper:=TRUE;
				END_IF

				tnWashing(IN:=xStartOper,  PT:= ((WORD_TO_TIME(wWashByWaterTime))*1000  - PauseOperationTime));
				wTimePassed:=REAL_TO_WORD(TIME_TO_REAL(tnWashing.ET)/1000) + wTimeBeforePause;
				wTimeOperationSet:=wWashByWaterTime;

				IF tnWashing.Q THEN
					tnWashing(IN:=FALSE);
					xStartOper:=FALSE;
					wTimePassed:=		0;
					PauseOperationTime:=T#0S;
					wTimeBeforePause:=0;
					(*
					IF xAlkaliCleaned THEN
						State:= EmptyAlkaliTank;
					ELSE
						State:=CheckAccid;
					END_IF
					*)
					IF xAlkaliCleaned THEN
						xAlkaliCleaned:=FALSE;
						wNextState:=FillAlkaliTank;
					ELSE
						wNextState:=CheckAccid;
					END_IF
					State:= EmptyAlkaliTank;
				END_IF


			FillAlkaliTank:



				xV_WaterOut:=		FALSE;
				xV_AlkaliIn:=			FALSE;
				xV_AlkaliOut:=			FALSE;
				xV_AllIn:=				FALSE;

				IF rAlkaliLevel >= wAlkaliLevelOK AND xAlkaliCooked AND xDissolvingStoped THEN
					IF xDoAccidTank THEN
						wNextState:=WashAccidTankWater;
						State:=EmptyAccidTank;
					ELSE
						xStart:=FALSE;
					END_IF
				END_IF




			EmptyAccidTank:



				xV_AccidOut:=				TRUE;
				xV_AlkaliOut:=				FALSE;
				xV_WaterOut:=			FALSE;
				xV_Drainage:=			FALSE;
				xV_UsedWaterInFill:=		FALSE;
				xV_AlkaliIn:=				FALSE;
				xV_AllIn:=					FALSE;
				xV_AccidIn:=				FALSE;

				IF (NOT xV_DrainageOn) AND xV_AccidOutOn THEN
					xPump:=TRUE;
				END_IF

				IF rAccidLevel < wAccidLevelDrain THEN
					xPump:=FALSE;
					xAcknawlage:=TRUE;
					State:= WaitManualAccidDrain;
				END_IF


			WaitManualAccidDrain:


				xPump:=				FALSE;
				xV_AccidOut:=				FALSE;
				xV_AlkaliIn:=			FALSE;
				xV_AllIn:=					FALSE;


				IF NOT xAcknawlage THEN
					(*
					IF XAccidCleaned THEN
						XAccidCleaned:=FALSE;
						xAcknawlage:=TRUE;
						State:= FillAccidTank;
					ELSE
					State:= WashAccidTankWater;
					END_IF
					*)
					State:=wNextState;
				END_IF



			WashAccidTankAlkali:


				xV_AllIn:=					TRUE;
				xV_Drainage_1:=			TRUE;
				xV_Drainage:=			TRUE;
				xV_AccidIn:=				TRUE;
				xV_AccidOut:=				FALSE;
				xV_AlkaliOut:=				TRUE;
				xV_WaterOut:=			FALSE;

				IF (NOT xV_AccidOutOn) AND xV_AllInOn AND xV_AccidInOn AND xV_AlkaliOutOn THEN
					xPump:=TRUE;
					xStartOper:=TRUE;
				END_IF

				tnWashing(IN:=xStartOper,  PT:= ((WORD_TO_TIME(wWashByAlkaliTime))*1000) - PauseOperationTime);
				wTimePassed:=REAL_TO_WORD(TIME_TO_REAL(tnWashing.ET)/1000) + wTimeBeforePause;
				wTimeOperationSet:=wWashByAlkaliTime;

				IF tnWashing.Q THEN
					tnWashing(IN:=FALSE);
					xStartOper:=FALSE;
					wTimePassed:=		0;
					PauseOperationTime:=T#0S;
					wTimeBeforePause:=0;
					XAccidCleaned:=TRUE;
					State:= WashAccidTankWater;
				END_IF



			WashAccidTankWater:


				xV_AllIn:=				TRUE;
				xV_Drainage_1:=		TRUE;
				xV_Drainage:=		TRUE;
				xV_AccidIn:=			TRUE;
				xV_WaterOut:=		TRUE;
				xV_AccidOut:=			FALSE;
				xV_AlkaliOut:=			FALSE;


				IF (NOT xV_AlkaliOutOn) AND xV_AllInOn AND xV_AccidInOn  THEN
					xPump:=TRUE;
					xStartOper:=TRUE;
				END_IF

				tnWashing(IN:=xStartOper,  PT:= ((WORD_TO_TIME(wWashByWaterTime))*1000) - PauseOperationTime);
				wTimePassed:=REAL_TO_WORD(TIME_TO_REAL(tnWashing.ET)/1000) + wTimeBeforePause;
				wTimeOperationSet:=wWashByWaterTime;

				IF tnWashing.Q THEN
					tnWashing(IN:=FALSE);
					xStartOper:=FALSE;

					wTimePassed:=		0;
					PauseOperationTime:=T#0S;
					wTimeBeforePause:=0;
					(*
					IF XAccidCleaned THEN
						State:= EmptyAccidTank;
					ELSE
						State:=CheckAlkali;
					END_IF
					*)
					IF XAccidCleaned THEN
						XAccidCleaned:=FALSE;
						wNextState:=FillAccidTank;
					ELSE
						wNextState:=CheckAlkali;
					END_IF
					State:= EmptyAccidTank;

				END_IF


			FillAccidTank:


				xV_Drainage_1:=		FALSE;
				xV_AccidIn:=			FALSE;
				IF rAccidLevel >= wAccidLevelOK AND xAccidCooked AND xDissolvingStoped AND (NOT xAcknawlage) THEN
					IF xDoAccidTank THEN
						xStart:=FALSE;
					END_IF
				END_IF


			CheckAlkali:


				IF rAlkaliLevel >= wAlkaliLevelOK  AND xDissolvingStoped THEN
					State:=WashAccidTankAlkali;
				ELSE
					xAcknawlage:= TRUE;
					State:= WaitAlkaliDissolving;
				END_IF



			WaitAlkaliDissolving:

				xV_AllIn:=					FALSE;
				IF rAlkaliLevel >= wAlkaliLevelOK  AND xDissolvingStoped AND (NOT xAcknawlage) THEN
					State:= WashAccidTankAlkali;
				END_IF


			CheckAccid:


				IF rAccidLevel >= wAccidLevelOK  AND xDissolvingStoped THEN
					State:=WashAlkaliTankAccid;
				ELSE
					(*
					xDoDissolveAccid:=TRUE;
					xStartDissolving:=TRUE;
					*)
					xAcknawlage:= TRUE;
					State:= WaitAccidDissolving;
				END_IF



			WaitAccidDissolving:

				IF rAccidLevel >= wAccidLevelOK AND xAccidCooked AND xDissolvingStoped AND (NOT xAcknawlage) THEN
					State:= WashAlkaliTankAccid;
				END_IF

END_CASE

IF NOT xStartOper THEN
	PauseOperationTime:=T#0S;
END_IF
END_FUNCTION_BLOCK

(* POU Process/SelfWashing/prSelfWashStateBits, ST *)
PROGRAM prSelfWashStateBits
VAR
END_VAR
SelfWashStateBits.0	:=	SelfWashState = 0	;
SelfWashStateBits.1	:=	SelfWashState = 1	;
SelfWashStateBits.2	:=	SelfWashState = 2	;
SelfWashStateBits.3	:=	SelfWashState = 3	;
SelfWashStateBits.4	:=	SelfWashState = 4	;
SelfWashStateBits.5	:=	SelfWashState = 5	;
SelfWashStateBits.6	:=	SelfWashState = 6	;
SelfWashStateBits.7	:=	SelfWashState = 7	;
SelfWashStateBits.8	:=	SelfWashState = 8	;
SelfWashStateBits.9	:=	SelfWashState = 9	;
SelfWashStateBits.10	:=	SelfWashState = 10	;
SelfWashStateBits.11	:=	SelfWashState = 11	;
SelfWashStateBits.12	:=	SelfWashState = 12	;
SelfWashStateBits.13	:=	SelfWashState = 13	;
SelfWashStateBits.14	:=	SelfWashState = 14	;
SelfWashStateBits.15	:=	SelfWashState = 15	;
SelfWashStateBits.16	:=	SelfWashState = 16	;
SelfWashStateBits.17	:=	SelfWashState = 17	;
SelfWashStateBits.18	:=	SelfWashState = 18	;
SelfWashStateBits.19	:=	SelfWashState = 19	;
SelfWashStateBits.20	:=	SelfWashState = 20	;
SelfWashStateBits.21	:=	SelfWashState = 21	;
SelfWashStateBits.22	:=	SelfWashState = 22	;
SelfWashStateBits.23	:=	SelfWashState = 23	;
SelfWashStateBits.24	:=	SelfWashState = 24	;
SelfWashStateBits.25	:=	SelfWashState = 25	;
SelfWashStateBits.26	:=	SelfWashState = 26	;
SelfWashStateBits.27	:=	SelfWashState = 27	;
SelfWashStateBits.28	:=	SelfWashState = 28	;
SelfWashStateBits.29	:=	SelfWashState = 29	;
SelfWashStateBits.30	:=	SelfWashState = 30	;
SelfWashStateBits.31	:=	SelfWashState = 31	;
SelfWashStateBits2.0	:=	SelfWashState = 32	;
SelfWashStateBits2.1	:=	SelfWashState = 33	;
SelfWashStateBits2.2	:=	SelfWashState = 34	;
SelfWashStateBits2.3	:=	SelfWashState = 35	;
SelfWashStateBits2.4	:=	SelfWashState = 36	;
SelfWashStateBits2.5	:=	SelfWashState = 37	;
SelfWashStateBits2.6	:=	SelfWashState = 38	;
SelfWashStateBits2.7	:=	SelfWashState = 39	;
SelfWashStateBits2.8	:=	SelfWashState = 40	;
SelfWashStateBits2.9	:=	SelfWashState = 41	;
SelfWashStateBits2.10	:=	SelfWashState = 42	;
SelfWashStateBits2.11	:=	SelfWashState = 43	;
SelfWashStateBits2.12	:=	SelfWashState = 44	;
SelfWashStateBits2.13	:=	SelfWashState = 45	;
SelfWashStateBits2.14	:=	SelfWashState = 46	;
SelfWashStateBits2.15	:=	SelfWashState = 47	;
SelfWashStateBits2.16	:=	SelfWashState = 48	;
END_PROGRAM

(* POU Process/Washing/prStateBits, ST *)
PROGRAM prStateBits
VAR
END_VAR
wWashingStateBitsLine1.0	:=	wWashingStateLine1 = 0	;
wWashingStateBitsLine1.1	:=	wWashingStateLine1 = 1	;
wWashingStateBitsLine1.2	:=	wWashingStateLine1 = 2	;
wWashingStateBitsLine1.3	:=	wWashingStateLine1 = 3	;
wWashingStateBitsLine1.4	:=	wWashingStateLine1 = 4	;
wWashingStateBitsLine1.5	:=	wWashingStateLine1 = 5	;
wWashingStateBitsLine1.6	:=	wWashingStateLine1 = 6	;
wWashingStateBitsLine1.7	:=	wWashingStateLine1 = 7	;
wWashingStateBitsLine1.8	:=	wWashingStateLine1 = 8	;
wWashingStateBitsLine1.9	:=	wWashingStateLine1 = 9	;
wWashingStateBitsLine1.10	:=	wWashingStateLine1 = 10	;
wWashingStateBitsLine1.11	:=	wWashingStateLine1 = 11	;
wWashingStateBitsLine1.12	:=	wWashingStateLine1 = 12	;
wWashingStateBitsLine1.13	:=	wWashingStateLine1 = 13	;
wWashingStateBitsLine1.14	:=	wWashingStateLine1 = 14	;
wWashingStateBitsLine1.15	:=	wWashingStateLine1 = 15	;
wWashingStateBitsLine1.16	:=	wWashingStateLine1 = 16	;
wWashingStateBitsLine1.17	:=	wWashingStateLine1 = 17	;
wWashingStateBitsLine1.18	:=	wWashingStateLine1 = 18	;
wWashingStateBitsLine1.19	:=	wWashingStateLine1 = 19	;
wWashingStateBitsLine1.20	:=	wWashingStateLine1 = 20	;
wWashingStateBitsLine1.21	:=	wWashingStateLine1 = 21	;
wWashingStateBitsLine1.22	:=	wWashingStateLine1 = 22	;
wWashingStateBitsLine1.23	:=	wWashingStateLine1 = 23	;
wWashingStateBitsLine1.24	:=	wWashingStateLine1 = 24	;
wWashingStateBitsLine1.25	:=	wWashingStateLine1 = 25	;
wWashingStateBitsLine1.26	:=	wWashingStateLine1 = 26	;
			
wWashingStateBitsLine2.0	:=	wWashingStateLine2 = 0	;
wWashingStateBitsLine2.1	:=	wWashingStateLine2 = 1	;
wWashingStateBitsLine2.2	:=	wWashingStateLine2 = 2	;
wWashingStateBitsLine2.3	:=	wWashingStateLine2 = 3	;
wWashingStateBitsLine2.4	:=	wWashingStateLine2 = 4	;
wWashingStateBitsLine2.5	:=	wWashingStateLine2 = 5	;
wWashingStateBitsLine2.6	:=	wWashingStateLine2 = 6	;
wWashingStateBitsLine2.7	:=	wWashingStateLine2 = 7	;
wWashingStateBitsLine2.8	:=	wWashingStateLine2 = 8	;
wWashingStateBitsLine2.9	:=	wWashingStateLine2 = 9	;
wWashingStateBitsLine2.10	:=	wWashingStateLine2 = 10	;
wWashingStateBitsLine2.11	:=	wWashingStateLine2 = 11	;
wWashingStateBitsLine2.12	:=	wWashingStateLine2 = 12	;
wWashingStateBitsLine2.13	:=	wWashingStateLine2 = 13	;
wWashingStateBitsLine2.14	:=	wWashingStateLine2 = 14	;
wWashingStateBitsLine2.15	:=	wWashingStateLine2 = 15	;
wWashingStateBitsLine2.16	:=	wWashingStateLine2 = 16	;
wWashingStateBitsLine2.17	:=	wWashingStateLine2 = 17	;
wWashingStateBitsLine2.18	:=	wWashingStateLine2 = 18	;
wWashingStateBitsLine2.19	:=	wWashingStateLine2 = 19	;
wWashingStateBitsLine2.20	:=	wWashingStateLine2 = 20	;
wWashingStateBitsLine2.21	:=	wWashingStateLine2 = 21	;
wWashingStateBitsLine2.22	:=	wWashingStateLine2 = 22	;
wWashingStateBitsLine2.23	:=	wWashingStateLine2 = 23	;
wWashingStateBitsLine2.24	:=	wWashingStateLine2 = 24	;
wWashingStateBitsLine2.25	:=	wWashingStateLine2 = 25	;
wWashingStateBitsLine2.26	:=	wWashingStateLine2 = 26	;
			
wWashingStateBitsLine3.0	:=	wWashingStateLine3 = 0	;
wWashingStateBitsLine3.1	:=	wWashingStateLine3 = 1	;
wWashingStateBitsLine3.2	:=	wWashingStateLine3 = 2	;
wWashingStateBitsLine3.3	:=	wWashingStateLine3 = 3	;
wWashingStateBitsLine3.4	:=	wWashingStateLine3 = 4	;
wWashingStateBitsLine3.5	:=	wWashingStateLine3 = 5	;
wWashingStateBitsLine3.6	:=	wWashingStateLine3 = 6	;
wWashingStateBitsLine3.7	:=	wWashingStateLine3 = 7	;
wWashingStateBitsLine3.8	:=	wWashingStateLine3 = 8	;
wWashingStateBitsLine3.9	:=	wWashingStateLine3 = 9	;
wWashingStateBitsLine3.10	:=	wWashingStateLine3 = 10	;
wWashingStateBitsLine3.11	:=	wWashingStateLine3 = 11	;
wWashingStateBitsLine3.12	:=	wWashingStateLine3 = 12	;
wWashingStateBitsLine3.13	:=	wWashingStateLine3 = 13	;
wWashingStateBitsLine3.14	:=	wWashingStateLine3 = 14	;
wWashingStateBitsLine3.15	:=	wWashingStateLine3 = 15	;
wWashingStateBitsLine3.16	:=	wWashingStateLine3 = 16	;
wWashingStateBitsLine3.17	:=	wWashingStateLine3 = 17	;
wWashingStateBitsLine3.18	:=	wWashingStateLine3 = 18	;
wWashingStateBitsLine3.19	:=	wWashingStateLine3 = 19	;
wWashingStateBitsLine3.20	:=	wWashingStateLine3 = 20	;
wWashingStateBitsLine3.21	:=	wWashingStateLine3 = 21	;
wWashingStateBitsLine3.22	:=	wWashingStateLine3 = 22	;
wWashingStateBitsLine3.23	:=	wWashingStateLine3 = 23	;
wWashingStateBitsLine3.24	:=	wWashingStateLine3 = 24	;
wWashingStateBitsLine3.25	:=	wWashingStateLine3 = 25	;
wWashingStateBitsLine3.26	:=	wWashingStateLine3 = 26	;
			
wWashingStateBitsLine4.0	:=	wWashingStateLine4 = 0	;
wWashingStateBitsLine4.1	:=	wWashingStateLine4 = 1	;
wWashingStateBitsLine4.2	:=	wWashingStateLine4 = 2	;
wWashingStateBitsLine4.3	:=	wWashingStateLine4 = 3	;
wWashingStateBitsLine4.4	:=	wWashingStateLine4 = 4	;
wWashingStateBitsLine4.5	:=	wWashingStateLine4 = 5	;
wWashingStateBitsLine4.6	:=	wWashingStateLine4 = 6	;
wWashingStateBitsLine4.7	:=	wWashingStateLine4 = 7	;
wWashingStateBitsLine4.8	:=	wWashingStateLine4 = 8	;
wWashingStateBitsLine4.9	:=	wWashingStateLine4 = 9	;
wWashingStateBitsLine4.10	:=	wWashingStateLine4 = 10	;
wWashingStateBitsLine4.11	:=	wWashingStateLine4 = 11	;
wWashingStateBitsLine4.12	:=	wWashingStateLine4 = 12	;
wWashingStateBitsLine4.13	:=	wWashingStateLine4 = 13	;
wWashingStateBitsLine4.14	:=	wWashingStateLine4 = 14	;
wWashingStateBitsLine4.15	:=	wWashingStateLine4 = 15	;
wWashingStateBitsLine4.16	:=	wWashingStateLine4 = 16	;
wWashingStateBitsLine4.17	:=	wWashingStateLine4 = 17	;
wWashingStateBitsLine4.18	:=	wWashingStateLine4 = 18	;
wWashingStateBitsLine4.19	:=	wWashingStateLine4 = 19	;
wWashingStateBitsLine4.20	:=	wWashingStateLine4 = 20	;
wWashingStateBitsLine4.21	:=	wWashingStateLine4 = 21	;
wWashingStateBitsLine4.22	:=	wWashingStateLine4 = 22	;
wWashingStateBitsLine4.23	:=	wWashingStateLine4 = 23	;
wWashingStateBitsLine4.24	:=	wWashingStateLine4 = 24	;
wWashingStateBitsLine4.25	:=	wWashingStateLine4 = 25	;
wWashingStateBitsLine4.26	:=	wWashingStateLine4 = 26	;
END_PROGRAM

(* POU Process/Washing/prWashingLine2, ST *)
PROGRAM prWashingLine2
VAR
	WashingProcess2:	fbWashingProcess;
	xResetErrors: BOOL;
	xPause: BOOL;
END_VAR
IF wDissolvingStateLine2 = 0 THEN
WashingProcess2(
	xReady:= (*xReadyForWashing AND*) wDissolvingStateLine2 = 0,
	arOperations:= arOperations,
	rWaterLevel:= CleanWaterLevel,
	rUsedWaterLevel:= UsedWaterLevel,
	rAccidLevel:= AccidLevel,
	rAlkaliLevel:= AlkaliLevel,
	wConcPumpTime:=arConcPumpTimeSteril[2, wChosenRecipeLine2],
	wConcMessureTime:= rConcCheckTime,
	arOperations2x:=arOperations2x,
	arOperations3x:=arOperations3x,
	wChosenRecipeLine:=wChosenRecipeLine2,
	wLine:=2,
	xPumpNorm:=Pump_InvNorm_2,

	rConcOfClkaliInTank:=rDissolAlkaliConcSet,
	rConcOfAccidInTank:=rDissolAccidConcSet,

	rWaterAfterSterilTime:=arWaterAfterSterilTime[2, wChosenRecipeLine2],
	wTafterAlkaliWater:=arTafterAlkaliWater[2, wChosenRecipeLine2],
	wTafterAccidWater:=arTafterAccidWater[2, wChosenRecipeLine2],

	rFlawWaterAfterAlcaliSet:=	arFlawWaterAfterAlcaliSet[2, wChosenRecipeLine2],
	rFlawWaterAfterAccidSet:=	arFlawWaterAfterAccidSet[2, wChosenRecipeLine2],
	rWaterAfterSterilFlaw:=	arWaterAfterSterilFlaw[2, wChosenRecipeLine2],
	rWaterAfterSterilConc:=	arWaterAfterSterilConc[2, wChosenRecipeLine2],
	rFlawWaterAfterAlcaliSet:=	arFlawWaterAfterAlcaliSet[2, wChosenRecipeLine2],
	rFlawWaterAfterAccidSet:=	arFlawWaterAfterAccidSet[2, wChosenRecipeLine2],
	wUsedWaterLevelOK:= wUsedWaterLevelOK,
	wUsedWaterLevelNotOK:= wUsedWaterLevelNotOK,
	wBackTget:= Heater_BackTget_2,
	xPause:= xPauseWashingLine2,
	xVoutOn:= xState_V211,
	xV_NotshortcutOn:= xState_V210,
	xV_UsedWaterInOn:= xState_V208,
	xV_AlkaliInOn:= xState_V206,
	xV_AccidInOn:= xState_V207,
	xV_WaterOutOn:= xState_V201,
	xV_UsedWaterOutOn:= xState_V202,
	xV_AlkaliOutOn:= xState_V204,
	xV_AccidOutOn:= xState_V203,
	xV_CycleOn:= xState_V205,
	xPumpOn:= Pump_OnAuto_2,
	rConcentration:= Conc_Line2,
	(*xAccidIsGoing:=xAccidIsGoing2,*)
	xFeedbackSwitch:= DI_FeedBackSwitchLine2,
	rWaterAfterSterilT:=arWaterAfterSterilT[2, wChosenRecipeLine2],
	wRecipeTimeRinse:= arWaterTime[2, wChosenRecipeLine2],
	wRecipeTimeAlcali:= arAlkaliTime[2, wChosenRecipeLine2],
	wRecipeTimeAccid:= arAccidTime[2, wChosenRecipeLine2],
	wAfterRinseConcAlk:= (*wAfterRinseConcAlk*)rConcSolutionStopoperationAlk,
	wAfterRinseConcAcc:= (*wAfterRinseConcAcc*)rConcSolutionStopoperationAcc,
	wAfterAlkWaterTime:= arAfterAlkaliWaterTime[2, wChosenRecipeLine2],
	wAfterAccWaterTime:= arAfterAccidWaterTime[2, wChosenRecipeLine2],
	rTwaterSet:= arTwaterSet[2, wChosenRecipeLine2],
	rTalcaliSet:= arTalkaliSet[2, wChosenRecipeLine2],
	rTaccidSet:= arTaccidSet[2, wChosenRecipeLine2],
	rConcAlcaliSet:= (*arConcAlkaliSet[2, wChosenRecipeLine2]*)rConcSolutionStartOperationAlk,
	rConcAccidSet:= (*arConcAccidSet[2, wChosenRecipeLine2]*)rConcSolutionStartOperationAcc,
	rFlawAlcaliSet:= arFlawAlkaliSet[2, wChosenRecipeLine2],
	rFlawWaterSet:= arFlawWaterSet[2, wChosenRecipeLine2],
	rFlawAccidSet:= arFlawAccidSet[2, wChosenRecipeLine2],
	wTsteril:= arTsterilSet[2, wChosenRecipeLine2],
	wFlawSteril:= arFlawSterilSet[2, wChosenRecipeLine2],
	rConcSteril:= arConcSterilSet[2, wChosenRecipeLine2],
	wSterilTime:= arSterilTime[2, wChosenRecipeLine2],
	wCountOfOperations:= 7,
	xStart:= xStartWashingLine2,
	xVout:= OnAuto_V211,
	xV_Notshortcut:= OnAuto_V210,
	xV_UsedWaterIn:= OnAuto_V208,
	xV_AlkaliIn:= OnAuto_V206,
	xV_AccidIn:= OnAuto_V207,
	xV_WaterOut:= OnAuto_V201,
	xV_UsedWaterOut:= OnAuto_V202,
	xV_AlkaliOut:= OnAuto_V204,
	xV_AccidOut:= OnAuto_V203,
	xV_Cycle:= OnAuto_V205,
	xV_Drainage:= OnAuto_V209,
	xPump:= Pump_OnAuto_2,
	xHeaterPower:= Heater_AutoSetT_2,
	xResetErrors:= xResetAlmAll,
	xPA:= PA_OnAuto_2,
	rToutSet:= Heater_AutoSetT_2,
	rFlawOutSet:= Pump_FlawAutoSet_2,
	xDone:=xWashingDone_Line2,
	State=> wWashingStateLine2,
	PauseState=> (*wWashingPauseStateLine2*),
	wTimePassed=> wWashingTimePassed2,
	wTimeOperationSet=> wWashingOperTimeSet2,
	wError=> wWashingErr_2);
END_IF
END_PROGRAM

(* POU Process/Washing/prWashingLine3, ST *)
PROGRAM prWashingLine3
VAR
	WashingProcess3:	fbWashingProcess;
	xResetErrors: BOOL;
END_VAR
IF wDissolvingStateLine3 = 0 THEN
WashingProcess3(
	xReady:= (*xReadyForWashing AND*) wDissolvingStateLine3 = 0,
	arOperations:= arOperations,
	rWaterLevel:= CleanWaterLevel,
	rUsedWaterLevel:= UsedWaterLevel,
	rAccidLevel:= AccidLevel,
	rAlkaliLevel:= AlkaliLevel,
	wConcPumpTime:=arConcPumpTimeSteril[3, wChosenRecipeLine3],
	wConcMessureTime:= rConcCheckTime,
	arOperations2x:=arOperations2x,
	arOperations3x:=arOperations3x,
	wChosenRecipeLine:=wChosenRecipeLine3,
	wLine:=3,
	rConcOfClkaliInTank:=rDissolAlkaliConcSet,
	rConcOfAccidInTank:=rDissolAccidConcSet,

	xPumpNorm:=Pump_InvNorm_3,

	rWaterAfterSterilTime:=arWaterAfterSterilTime[3, wChosenRecipeLine3],
	wTafterAlkaliWater:=arTafterAlkaliWater[3, wChosenRecipeLine3],
	wTafterAccidWater:=arTafterAccidWater[3, wChosenRecipeLine3],

